SAVE: T     #S_SOFT; // Softwareschalter schreiben
NE3:  NOP   0;
NETWORK
TITLE =FC-Ausgang Q1

      U     #lb_Q1;
      =     #Q1;
NETWORK
TITLE =FC-Ausgang Q2

      U     #lb_Q2;
      =     #Q2;
NETWORK
TITLE =FC-ENO-Ausgang = Schaltausgang, für direkte FC-Verknüfpung

      O     #lb_Q1; // Ausgang 1
      O     #lb_Q2; // Ausgang 2
      SAVE  ; // auf FC-ENO-Ausgang geben
      CLR   ;

NETWORK
TITLE =Lokalen Speicher wieder in dauerhaften Zwischenspeicher

      L     LB     0;
      T     #bTmp;
      NOP   0;
END_FUNCTION

FUNCTION "m7b_udtCopyArray" : VOID
TITLE =kopiert einzelne UDT's von UDT-Arrays
//Kopiert UDT's aus Arrays, die Datenlänge des UDT wird automatisch ermittelt.
//Anpassungen der Datenlänge nach Änderungen an den UDT's entfällt somit.
//
//Achtung Array bzw. Speichergrenzen werden nicht überprüft.
//Gegebenenfalls, Indexangaben vorher auf Korrektheit prüfen bzw. limittieren!
//Bei inkorrekten Indexangaben geht CPU in STOP.
//
//Verwendung: Verwaltung von Datensätzen wie Rezepturen, Betriebsdaten,
//Positionsdaten usw. in der Steuerung.
//
//Kopiert wird von/zu: DB, statischen Lokaldaten im Instanz-DB
//(Multinnstanzfähig, ohne zus. Adresskorrektur, da Step7 bei Verwendung von
//Instanzdaten bei UDT's automatisch als Quelle [#84] DB und Nr. mit korrekter
//Adress angibt statt nur DI [#85])
//
//Nicht kopiert wrid von/zu lokalen Daten (TEMP), da vor- vorherige Lokaldaten
//benötigt werden (S7 aber nur vorherige Lokaldaten unterstützt)
//
//[IN]
//srcUdtArray : Anypointer auf den ersten UDT im Quell-Array
//srcIndex    : Index des Quell-UDT im Array, beginnend bei 0
//destUdtArray: Anypointer auf den ersten UDT im Ziel-Array
//destIndex   : Index des Ziel-UDT im Array, beginnend mit 0
//
//AUTOR: Stefan Maag, Dipl.-Ing. (FH) Elektrotechnik
//DATUM: 10/2007
//INTERNET: www.maagic7.de
//
//AENDERUNGSVERMERKE:
//--------------------------------------------------------------------------------
//DATUM        NAME       AENDERUNG
//--------------------------------------------------------------------------------
//20.03.2017   S.Maag     Verwendung von AR2 entfernt und Abfrage auf
//                        Daten Speicherbereich #87 vorheriger Lokaldatenstack
//                        hinzugefügt, da Daten aus vorherigem Stack nicht
//                        kopiert werden können, da BLKMOVE neuen L-Stack anlegt
//--------------------------------------------------------------------------------
//
AUTHOR : 'S.Maag'
FAMILY : Maagic7
VERSION : 0.1


VAR_INPUT
  srcUdtArray : ANY ;
  srcIndex : INT ;
  destUdtArray : ANY ;
  destIndex : INT ;
END_VAR
VAR_OUTPUT
  BLKMOV_RetVal : INT ;	//Return Value der Blockmovefunktion
END_VAR
VAR_TEMP
  pSRC : ANY ;	//mit Indexdaten modifizierter Quellpointer für BlockMove-Funktion
  pDEST : ANY ;	//mit Indexdaten modifizierter Zielpointer für BlockMove-Funktion
  dwPart1 : DWORD ;
  wPart2 : WORD ;
  dwPart3_Address : DWORD ;
  dwBitAddress : DWORD ;
  bMemory : BYTE ;	//Speicherbereich
END_VAR
BEGIN
NETWORK
TITLE =
//ANY
//Byte 0: 10h für S7
//Byte 1: Datentyp
//Byte 2..3: Wiederholungsfaktor
//Byte 4..5: DB-Nr
//Byte 6: Speicherbereich
//Byte 7..9: Byte/Bit-Adresse
//
//Speicherbereiche
//#80  P : Perepherie
//#81  E : Eingänge
//#82  A : Ausgänge
//#83  M : Merker
//#84  DB : Datenbaustein
//#85  DI : Instanz-DB
//#86  L  : Lokaldaten (L-Stack)
//#87  V  : Verherige Lokaldaten


NETWORK
TITLE =ANY-Pointer Quelle für BlockMove bearbeiten
//Beim Wiederholungsfaktor wird automatisch von Byte ausgegeangen.
//Für UDT's stimmt dies auch immer. Falls der Baustein allgemein zum kopieren von
//Anypointerbasierten Daten verwendet werden soll, so muss dies beachtet bzw.
//angepasst werden.
//Den ANY-Pointer Quelle mit den Indexdaten modifizieren und als ANY-Pointer für
//die BlockMove-Funktion speichern
      L     P##srcUdtArray; // Pointer auf den Quellpointer
      LAR1  ; // in Adressregister 1

      L     D [AR1,P#0.0]; // Part1
      T     #dwPart1;
      L     W [AR1,P#4.0]; // Part2
      T     #wPart2;
      L     D [AR1,P#6.0]; // Part3  (Address-Pointer)
      T     #dwPart3_Address;
      SRD   24; // Shift 3 Byte = Speicherbereich
      T     #bMemory;
      L     B#16#87; // Daten vom vorherigen Lockaldaten Stack (geht nicht!)
      ==I   ;
      SPB   ERR;


// Calculating the Address with Source ARRAY Index
      L     W [AR1,P#2.0]; // Wiederholungsfaktor
      L     #srcIndex;
      *I    ; // Offset aus Index für Quellbereich
      SLD   3; // ins Pointerformat konvertieren
      L     #dwPart3_Address; // Ursprüngliche Quelladdresse
      UD    DW#16#FFFFFF; // oberes Byte fuer Speicherbereich ausblenden
      +D    ; // Quelladresspointer mit verrechnetem Index
      T     #dwBitAddress;

      L     P##pSRC; // Pointer auf AnyPointer Quelle für BlockMove
      LAR1  ; // in Adressreguster 1

      L     #dwPart1; // Part 1 of ANY
      T     D [AR1,P#0.0]; // to pSRC [ANY]

      L     #wPart2; // Part 2
      T     W [AR1,P#4.0]; // DB-Nr.

      L     #dwPart3_Address; // Part 3 Address
      UD    DW#16#FF000000; // Speicherbereich maskieren
      L     #dwBitAddress; // mit Array-Index modifizierte Adresse
      OD    ; // Speicherbereich_Adresse zusammenführen
      T     D [AR1,P#6.0];

NETWORK
TITLE =ANY-Pointer Ziel für BlockMove bearbeiten

      L     P##destUdtArray; // Pointer auf den Quellpointer
      LAR1  ; // in Adressregister 1

      L     D [AR1,P#0.0]; // Part1
      T     #dwPart1;
      L     W [AR1,P#4.0]; // Part2
      T     #wPart2;
      L     D [AR1,P#6.0]; // Part3  (Address-Pointer)
      T     #dwPart3_Address;
      SRD   24; // Shift 3 Byte = Speicherbereich
      T     #bMemory;
      L     B#16#87; // Daten vom vorherigen Lockaldaten Stack (geht nicht!)
      ==I   ;
      SPB   ERR;

// Calculating the Address with Destination ARRAY Index
      L     W [AR1,P#2.0]; // Wiederholungsfaktor
      L     #destIndex;
      *I    ; // Offset aus Index für Quellbereich
      SLD   3; // ins Pointerformat konvertieren
      L     #dwPart3_Address; // Ursprüngliche Quelladdresse
      UD    DW#16#FFFFFF; // oberes Byte fuer Speicherbereich ausblenden
      +D    ; // Quelladresspointer mit verrechnetem Index
      T     #dwBitAddress;

      L     P##pDEST; // Pointer auf AnyPointer Quelle für BlockMove
      LAR1  ; // in Adressreguster 1

      L     #dwPart1; // Part 1 of ANY
      T     D [AR1,P#0.0]; // to pDEST [ANY]

      L     #wPart2; // Part 2
      T     W [AR1,P#4.0]; // DB-Nr.

      L     #dwPart3_Address; // Part 3 Address
      UD    DW#16#FF000000; // Speicherbereich maskieren
      L     #dwBitAddress; // mit Array-Index modifizierte Adresse
      OD    ; // Speicherbereich_Adresse zusammenführen
      T     D [AR1,P#6.0];

NETWORK
TITLE =kopieren der Daten mittels BlockMove

      CALL "BLKMOV" (
           SRCBLK                   := #pSRC,
           RET_VAL                  := #BLKMOV_RetVal,
           DSTBLK                   := #pDEST);
      NOP   0;
NETWORK
TITLE =

      SET   ;
      SAVE  ;
      BEA   ;

NETWORK
TITLE =
//Daten vom vorherigen Lokaldatenstack können nicht kopiert werden, da
//BLKMOVE neuen L-Stack öffnet und die Daten somit vom vor- vorherigen Stack
//wären
ERR:  L     W#16#8888; // Daten vom vorheriger Lockaldatenstack
      T     #BLKMOV_RetVal; // können nicht kopiert werden, da BLKMOVE neuen Stack anlegt
      SET   ;
      SAVE  ;
      BE    ;

END_FUNCTION

FUNCTION "m7b_MultiEventCounter" : VOID
TITLE =Multi-Ereigniszähler mit GesamtAnzahl im Ereignis 0
//Zähler für verschiedene Ereignisse. Es wird immer jeweils bei einem Zählvorgang
//der entsprechende Ereigniszähler und der Gesamtzähler erhöht. Eine Überprüfung
//auf die Gültigkeit des übergebenen DBs und richtige Länge wird nicht
//druchgeführt.
//
//AUTOR: Stefan Maag, Dipl.-Ing. (FH) Elektrotechnik
//DATUM: 5/2003
//INTERNET: www.maagic7.de
//
//AENDERUNGSVERMERKE:
//--------------------------------------------------------------------------------
//DATUM        NAME            AENDERUNG
//--------------------------------------------------------------------------------
//
//--------------------------------------------------------------------------------
//
//HINWEISE:
AUTHOR : 'S.Maag'
FAMILY : Maagic7
VERSION : 0.1


VAR_INPUT
  DBNr : INT ;	//Nr des Datenbausteins für Zählereignisse
  StartAdr : INT ;	//StartAdr. des ersten Eintrags
  EventNr : INT ;	//Nr des zu zählenden Ereignisses; Nr.0 = Gesamtzaehler
  Count : BOOL ;	//Befehl zählen
END_VAR
VAR_TEMP
  tmpDB : INT ;
  tmpPtrOff : INT ;
  AR1 : DWORD ;
END_VAR
BEGIN
NETWORK
TITLE =Überprüfung auf Zählen!

      UN    #Count;
      BEB   ;
NETWORK
TITLE =ungültige EreignisNr - ENDE

      L     #EventNr;
      L     1;
      <I    ;
      BEB   ;
NETWORK
TITLE =DB öffnen und Pointer auf StartAdresse erzeugen

      TAR1  #AR1; // Adressregister 1 sichern

      L     #DBNr;
      T     #tmpDB;

      AUF   DB [#tmpDB];

      L     #StartAdr; // Startadresse ins Pointerformat
      SLD   3;
      TAR1  ; // ins Adressregister 1

NETWORK
TITLE =GesamtZaehler bearbeiten


      L     DBD [AR1,P#0.0]; // Gesamtzählerstand aus DB lesen
      +     1;
      T     DBD [AR1,P#0.0]; // neuen Gesamtzählerstand speichern

NETWORK
TITLE =Pointer Auf EreignisZähler-Daten erzeugen

      TAR1  ; // Pointer auf Startadresse in Akku 1 zurueck
      L     #EventNr; // EreignisNr
      SLD   5; // EreignisNr -> BitPointer (*16; DINT=32Bit)
      +D    ; // Pointer aus Ereignis zum StartPointer addieren
      LAR1  ; // Pointer auf EreignisZähler nach Adressregister 1

NETWORK
TITLE =EreignisZähler bearbeiten

      L     DBD [AR1,P#0.0]; // Ereigniszählerstand aus DB lesen
      +     1;
      T     DBD [AR1,P#0.0]; // neuen Ereigniszählerstand speichern

NETWORK
TITLE =FC-ENO Ausgang

      LAR1  #AR1; // ursprüngliches Adressregister 1 herstellen
      SET   ;
      SAVE  ;
      CLR   ;

END_FUNCTION

FUNCTION "m7b_udtCompareArray" : VOID
TITLE =udt Daten in Arrays vergleichen
//Vergleicht UDT's aus Arrays, die Datenlänge des UDT wird automatisch ermittelt.
//Anpassungen der Datenlänge nach Änderungen an den UDT's entfällt somit.
//
//Achtung!
//   Array bzw. Speichergrenzen werden nicht überprüft.
//   Gegebenenfalls, Indexangaben vorher auf Korrektheit prüfen bzw. limittieren!
//   Bei inkorrekten Indexangaben geht CPU in STOP.
//
//   Bei Verwendung von Strings in UDT's kann es vorkommen, dass zwischen dem
//   letzten Zeichen und reservierter Stringlänge noch tote Bytes mit
//   undefinierten Werten liegen. Dann ergibt der Vergleich des UDT ungleich, ein
//   Stringvergleich würde jedoch gleich ergeben.
//
//Verwendung: Verwaltung von Datensätzen wie Rezepturen, Betriebsdaten,
//Positionsdaten usw. in der Steuerung.
//
//[IN]
//srcUdtArray : Anypointer auf den ersten UDT im Quell-Array
//srcIndex    : Index des Quell-UDT im Array, beginnend bei 0
//cmpUdtArray : Anypointer auf den ersten UDT im Vergleichs-Array
//cmpIndex    : Index des Vergleichs-UDT im Array, beginnend mit 0
//
//[RET]
//ENO         : True if datas are equal
//
//AUTOR: Stefan Maag, Dipl.-Ing. (FH) Elektrotechnik
//DATUM: 10/2010
//INTERNET: www.maagic7.de
//
//AENDERUNGSVERMERKE:
//--------------------------------------------------------------------------------
//DATUM        NAME            AENDERUNG
//--------------------------------------------------------------------------------
//
//--------------------------------------------------------------------------------
//
//HINWEISE: AR2, Global- und Instanz DB muessen nicht gesichert werden, da diese
//           bei Call Aufrufen automatisch vom System wieder hergestellt werden.
//          (Bei UC Aufrufen nicht!)
//
//Vergleichroutine basiert auf m7b_DB_COMPARE_ByRef FC218
AUTHOR : 'S.Maag'
FAMILY : Maagic7
VERSION : 0.1


VAR_INPUT
  srcUdtArray : ANY ;
  srcIndex : INT ;
  cmpUdtArray : ANY ;
  cmpIndex : INT ;
END_VAR
VAR_TEMP
  AR1 : DWORD ;
  p_srcData : DWORD ;
  p_cmpData : DWORD ;
  srcRepeat : WORD ;
  cmpRepeat : WORD ;
  srcDataType : BYTE ;
  cmpDataType : BYTE ;
  srcDB_No : WORD ;
  cmpDB_no : WORD ;
  DB_NO : WORD ;
  srcSpeicherBereich : BYTE ;
  cmpSpeicherBereich : BYTE ;
  LOOPS : INT ;
  NoOfBytes : INT ;
  srcIsDB : BOOL ;
  cmpIsDB : BOOL ;
  pTest : DWORD ;
END_VAR
BEGIN
NETWORK
TITLE =Adressregiste 1 sichern
//Adressregister 2 Global- und Instanz DB werden bei CALL-Aufrufen automatisch
//vom System gesichert, bei UC nicht!
      TAR1  #AR1; // Adressregister 1 sichern

NETWORK
TITLE =Adressdaten aus ANY-Pointer extrahieren
//Beim Wiederholungsfaktor wird automatisch von Byte ausgegeangen.
//Für UDT's stimmt dies auch immer. Falls der Baustein allgemein zum vergleichen
//von Anypointerbasierten Daten verwendet werden soll, so muss dies beachtet bzw.
//angepasst werden.
//
      L     P##srcUdtArray; // Pointer auf den Quellpointer
      LAR1  ; // in Adressregister 1

      L     B [AR1,P#1.0]; // Byte 1 = Datentyp
      T     #srcDataType;

      L     B [AR1,P#6.0]; // Byte 6 = Speicherbereich
      T     #srcSpeicherBereich;

      L     W [AR1,P#4.0]; // DB-Nummer oder 0, wenn kein DB
      T     #srcDB_No;

      L     W [AR1,P#2.0]; // Wiederholungsfaktor
      T     #srcRepeat;
      L     #srcIndex;
      *I    ; // Offset aus Index für Quellbereich
      SLD   3; // ins Pointerformat konvertieren
      L     D [AR1,P#6.0]; // DatenAdresse im Pointeformat aus ANY
      +D    ; // Adresspointer mit verrechnetem Index
      T     #p_srcData; // Pointer Source Data

      L     P##cmpUdtArray; // Pointer auf Vergleichs UDT
      LAR1  ; // in Adressregister 1

      L     B [AR1,P#1.0]; // Byte 1 = Datentyp
      T     #cmpDataType;

      L     B [AR1,P#6.0]; // Byte 6 = Speicherbereich
      T     #cmpSpeicherBereich;

      L     W [AR1,P#4.0]; // DB-Nummer oder 0, wenn kein DB
      T     #cmpDB_no;

      L     W [AR1,P#2.0]; // Wiederholungsfaktor
      T     #cmpRepeat;
      L     #cmpIndex;
      *I    ; // Offset aus Index für Vergleichsbereich
      SLD   3; // ins Pointerformat konvertieren
      L     D [AR1,P#6.0]; // DatenAdresse im Pointeformat aus ANY
      +D    ; // Adresspointer mit verrechnetem Index
      T     #p_cmpData; // Pointer Vergleichsdaten

NETWORK
TITLE =Prüfen ob gleiches Datenformat, wenn NEIN, dann Daten ungleich
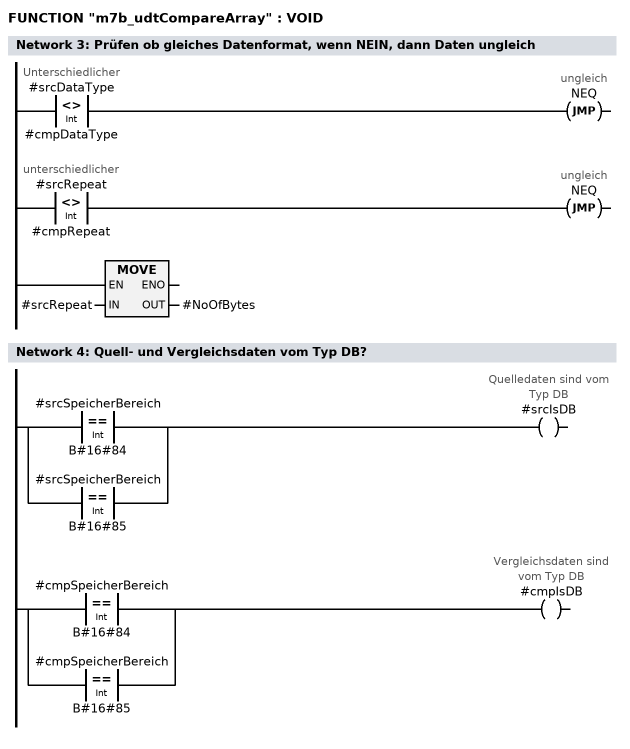

      L     #srcDataType; // Unterschiedlicher
      L     #cmpDataType; // Datentyp?
      <>I   ;
      SPB   NEQ; // ungleich

      L     #srcRepeat; // unterschiedlicher
      L     #cmpRepeat; // Wiederholungsfaktor
      <>I   ;
      SPB   NEQ; // ungleich

      L     #srcRepeat; // srcRepeat=cmpRepeat, deshalb
      T     #NoOfBytes; // Anzahl zu vergleichender Bytes gleich

NETWORK
TITLE =Quell- und Vergleichsdaten vom Typ DB?

      O(    ;
      L     #srcSpeicherBereich;
      L     B#16#84; // Datenbaustein
      ==I   ;
      )     ;
      O(    ;
      L     #srcSpeicherBereich;
      L     B#16#85; // Instanzdatenbaustein
      ==I   ;
      )     ;
      =     #srcIsDB; // Quelledaten sind vom Typ DB

      O(    ;
      L     #cmpSpeicherBereich;
      L     B#16#84; // Datenbaustein
      ==I   ;
      )     ;
      O(    ;
      L     #cmpSpeicherBereich;
      L     B#16#85; // Instanzdatenbaustein
      ==I   ;
      )     ;
      =     #cmpIsDB; // Vergleichsdaten sind vom Typ DB

NETWORK
TITLE =Vorbereitung für Vergleichsroutine
//Für die eigentliche Vergleichsroutine ist es nur relevant ob die Daten aus
//einem DB stammen, nicht ob Instanz oder Global-DB. Für den vergleich wird
//temporär immer ein DB als Global-DB, der andere als Instanz-DB geöffnet. Da dies
// nur nach Nummern geschieht, ist es egal welcher der DBs wie geöffnet wird.
//Codierung Speicherbereich:
//80h : P : Peripherie
//81h : E : Eingänge
//82h : A : Ausgänge
//83h : M : Merker
//84h : DB: Datenbaustein
//85h : DI: Instanzdatenbaustein
//86h : L : Lokaldaten (L-Stack)
//87h : V : voriger Lokaldatenstack
      UN    #srcIsDB; // Wenn weder Qell noch Vergleichsdaten
      UN    #cmpIsDB; // vom Typ DB
      SPB   DO; // dann keine Modifikation der DB-Kennung nötig, sofort vergleichen

      UN    #srcIsDB; // Wenn Quell-Daten nicht aus DB dann weiter,
      SPB   w1; // sonst Global-DB Kennung in Quelldatenpointer eintragen

      LAR1  P##p_srcData; // Adressregister 1 mit Pointer auf p_srcData laden
      L     B#16#84; // Wert für Global-DB-Kennung
      T     B [AR1,P#0.0]; // 84h=DB in p_srcData als Speicherbereichskennung eintragen

      AUF   DB [#srcDB_No]; // Datenbaustein Quelldaten als Global-DB öffnen

w1:   UN    #cmpIsDB; // Wenn Vergleichs-Daten nicht aus DB dann weiter,
      SPB   save; // sonst Instanz-DB Kennung in Quelldatenpointer eintragen

      LAR1  P##p_cmpData; // Adressregister 1 mit Pointer auf p_cmpData laden
      L     B#16#85; // Wert für Instanz-DB-Kennung
      T     B [AR1,P#0.0]; // 85h=DB in p_srcData als Speicherbereichskennung eintragen

      AUF   DI [#cmpDB_no]; // Datenbaustein Vergleichsdaten als Instanz-DB öffnen

save: L     #p_srcData; // Pointer der Quelldaten p_srcData in Adressregister 1
      LAR1  ;
      L     #p_cmpData; // Pointer der Vergleichsdaten p_cmpData in Adressregister 2
      LAR2  ;
NETWORK
TITLE =Vergleich der Daten
//Vergleich der Daten
//Vergleichroutine basiert auf m7b_DB_COMPARE_ByRef FC218
DO:   L     #NoOfBytes; // Anzahl der zu vergleichenden Bytes
      L     4; // in Anzahl der 32-Bit-Werte umrechen
      /I    ;
      SPZ   bts; // Wenn 0 32-Bit Werte, dann weiter mit letzten 3 Bytes
LOOP: T     #LOOPS;
      L     D [AR1,P#0.0]; // QuellDaten lesen
      L     D [AR2,P#0.0]; // VergleichsDaten lesen
      <>D   ; // wenn nicht gleich, dann Ende
      SPB   NEQ;
      +AR1  P#4.0; // Quell-Pointer in AR1 um 4 Bytes erhöhen
      +AR2  P#4.0; // Vergleichs-Pointer in AR2 um 4 Bytes erhöhen
      L     #LOOPS; // Schleifenzähler wieder in Akku 1 zurück
      LOOP  LOOP; // Schleifenzähler bearbeiten

bts:  L     #NoOfBytes; // nun noch die evtl. letzte 3 Bytes prüfen
      L     2#11; // Anzahl übriger Bytes maskieren
      UW    ; // Anzahl übriger Bytes
      SPZ   EQ; // Wenn 0 dann ENDE
LOP1: T     #LOOPS;
      L     B [AR1,P#0.0]; // QuellDaten lesen
      L     B [AR2,P#0.0]; // VergleichsDaten lesen
      <>I   ; // wenn nicht gleich, dann Ende
      SPB   NEQ;
      +AR1  P#1.0; // Quell-Pointer in AR1 um 1 Bytes erhöhen
      +AR2  P#1.0; // Vergleichs-Pointer in AR2 um 1 Bytes erhöhen
      L     #LOOPS; // Schleifenzähler wieder in Akku 1 zurück
      LOOP  LOP1; // Schleifenzähler bearbeiten

EQ:   SET   ; // Daten sind gleich (equal)
      SAVE  ;
      CLR   ;
      SPA   END;

NEQ:  CLR   ; // Daten sind ungleich (not equal)
      SAVE  ;

NETWORK
TITLE =Adressregister 1 wieder herstellen

END:  LAR1  #AR1; // ursprüngliches Adressregister 1 herstellen


END_FUNCTION

FUNCTION "m7b_2xSTART_SWITCH" : VOID
TITLE =2-fach Startumschalter
//Dieser Baustein ermöglicht, 2 Geräte (z.B. Kompressoren) abwechselnd
//einzuschalten. Dazu werden bei jedem Ausschalten eines Gerätes die beiden
//FRG-Ausgänge des Bausteins umgeschaltet.
//
//Verwendung: Startumschaltung von Kompressorenpaaren bei Klimaanlagen
//
//AUTOR: Stefan Maag, Dipl.-Ing. (FH) Elektrotechnik
//DATUM: 4/2004
//INTERNET: www.maagic7.de
//
//AENDERUNGSVERMERKE:
//--------------------------------------------------------------------------------
//DATUM        NAME            AENDERUNG
//--------------------------------------------------------------------------------
//
//--------------------------------------------------------------------------------
//
//HINWEISE:
AUTHOR : 'S.Maag'
FAMILY : Maagic7
VERSION : 0.1


VAR_INPUT
  G1_RUN : BOOL ;	//Eingang Gerät 1 läuft
  G2_RUN : BOOL ;	//Eingang Gerät 2 läuft
END_VAR
VAR_OUTPUT
  FRG1 : BOOL ;	//Freigabe Start Gerät 1
  FRG2 : BOOL ;	//Freigabe Start Gerät 2
END_VAR
VAR_IN_OUT
  bTMP : BYTE ;	//statisches Hilfsbyte
END_VAR
VAR_TEMP
  lb_SWITCH : BOOL ;	//Bit 0 von IO-Byte bTMP : Umschalter
  lb_FN : BOOL ;	//Negative Flanke Geräte ausgeschaltet
  lb2 : BOOL ;
  lb3 : BOOL ;
  lb4 : BOOL ;
  lb5 : BOOL ;
  lb6 : BOOL ;
  lb7 : BOOL ;	//Bit 7 von IO-Byte bTMP
END_VAR
BEGIN
NETWORK
TITLE =statisches HilfsByte in Lokaldatenbereich

      L     #bTMP;
      T     LB     0;
      NOP   0;
NETWORK
TITLE =Freigabe umschalten, wenn beide Geräte aus sind

      O     #G1_RUN;
      O     #G2_RUN;
      FN    #lb_FN;
      SPBN  NE2;
      UN    #lb_SWITCH;
      =     #lb_SWITCH;
NE2:  NOP   0;
NETWORK
TITLE =Bausteinausgang Freigabe Gerät 1

      UN    #lb_SWITCH;
      =     #FRG1;

NETWORK
TITLE =Bausteinausgang Freigabe Gerät 2

      U     #lb_SWITCH;
      =     #FRG2;

NETWORK
TITLE =statisches HilfsByte aus Lokaldatenbereich zurück

      L     LB     0;
      T     #bTMP;
      NOP   0;
NETWORK
TITLE =

      SET   ;
      SAVE  ;
      CLR   ;


END_FUNCTION

FUNCTION "m7b_MSG_2_ML" : VOID
TITLE =Meldungen (16Stk) mittels 2er Meldeleuchten anzeigen
//AUTOR: Stefan Maag, Dipl.-Ing. (FH) Elektrotechnik
//DATUM: 04/2006
//INTERNET: www.maagic7.de
//
//AENDERUNGSVERMERKE:
//--------------------------------------------------------------------------------
//DATUM        NAME      AENDERUNG
//--------------------------------------------------------------------------------
//
//--------------------------------------------------------------------------------
//
//HINWEISE:
AUTHOR : 'S.Maag'
FAMILY : Maagic7
VERSION : 0.1


VAR_INPUT
  MSG_1_8 : BYTE ;	//Meldung 1 bis 8 als Bits
  MSG_9_16 : BYTE ;
  TAKT_BYTE : BYTE ;	//System Taktmerkerbyte
END_VAR
VAR_OUTPUT
  ML1 : BOOL ;
  ML2 : BOOL ;
END_VAR
VAR_TEMP
  MSG_1 : BOOL ;
  MSG_2 : BOOL ;
  MSG_3 : BOOL ;
  MSG_4 : BOOL ;
  MSG_5 : BOOL ;
  MSG_6 : BOOL ;
  MSG_7 : BOOL ;
  MSG_8 : BOOL ;
  MSG_9 : BOOL ;
  MSG_10 : BOOL ;
  MSG_11 : BOOL ;
  MSG_12 : BOOL ;
  MSG_13 : BOOL ;
  MSG_14 : BOOL ;
  MSG_15 : BOOL ;
  MSG_16 : BOOL ;
  TAKT_100 : BOOL ;
  TAKT_200 : BOOL ;
  TAKT_400 : BOOL ;
  TAKT_500 : BOOL ;
  TAKT_800 : BOOL ;
  TAKT_1000 : BOOL ;
  TAKT_1600 : BOOL ;
  TAKT_2000 : BOOL ;
END_VAR
BEGIN
NETWORK
TITLE =Meldungsbits für Einzelbitverarbeitung in Lokaldatenbereich

      L     #MSG_1_8;
      T     LB     0;

      L     #MSG_9_16;
      T     LB     1;

      L     #TAKT_BYTE;
      T     LB     2;

      L     LW     0; // Alle 16 Meldungsbits laden
      L     0; // und auf 0 prüfen
      ==I   ; // wenn 0, dann keine Meldung
      SPB   E0; // keine Meldung

NETWORK
TITLE =Meldung nach Priorität auswählen
//Durch vertauschen der Auswertungen und Sprünge kann die Priortät der
//angezeigten Meldungen in gewünschter Reihenfolge festgelegt werden
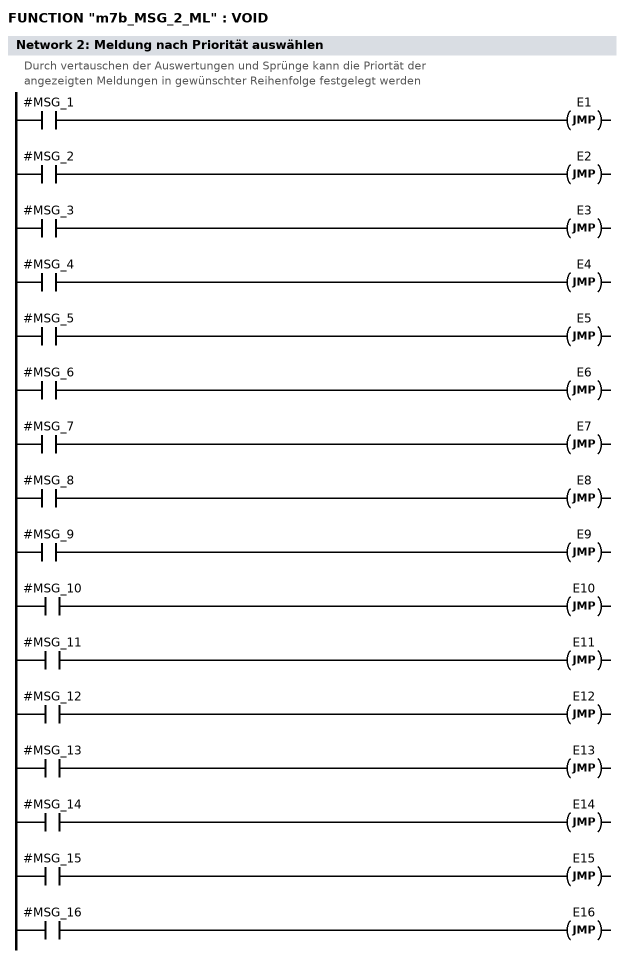
      U     #MSG_1;
      SPB   E1;
      U     #MSG_2;
      SPB   E2;
      U     #MSG_3;
      SPB   E3;
      U     #MSG_4;
      SPB   E4;
      U     #MSG_5;
      SPB   E5;
      U     #MSG_6;
      SPB   E6;
      U     #MSG_7;
      SPB   E7;
      U     #MSG_8;
      SPB   E8;
      U     #MSG_9;
      SPB   E9;
      U     #MSG_10;
      SPB   E10;
      U     #MSG_11;
      SPB   E11;
      U     #MSG_12;
      SPB   E12;
      U     #MSG_13;
      SPB   E13;
      U     #MSG_14;
      SPB   E14;
      U     #MSG_15;
      SPB   E15;
      U     #MSG_16;
      SPB   E16;

NETWORK
TITLE =Meldungen 0..3: ML2=AUS

E0:   CLR   ; // keine Störung
      =     #ML1;
      SPA   M0;

E1:   U     #TAKT_1000;
      =     #ML1;
      SPA   M0;

E2:   U     #TAKT_400;
      =     #ML1;
      SPA   M0;

E3:   SET   ;
      =     #ML1;

M0:   CLR   ;
      =     #ML2;
      SPA   END;

NETWORK
TITLE =Meldungen 4..7: ML2=TAKT_400ms

E4:   CLR   ;
      =     #ML1;
      SPA   M1;

E5:   U     #TAKT_1000;
      =     #ML1;
      SPA   M1;

E6:   U     #TAKT_400;
      =     #ML1;
      SPA   M1;

E7:   SET   ;
      =     #ML1;

M1:   U     #TAKT_1000;
      =     #ML2;
      SPA   END;

NETWORK
TITLE =Meldungen 8..11: ML2=TAKT_1000ms

E8:   CLR   ;
      =     #ML1;
      SPA   M2;

E9:   U     #TAKT_1000;
      =     #ML1;
      SPA   M2;

E10:  U     #TAKT_400;
      =     #ML1;
      SPA   M2;

E11:  SET   ;
      =     #ML1;

M2:   U     #TAKT_400;
      =     #ML2;
      SPA   END;

NETWORK
TITLE =Meldungen 12..15: ML2=EIN

E12:  CLR   ;
      =     #ML1;
      SPA   M3;

E13:  U     #TAKT_1000;
      =     #ML1;
      SPA   M3;

E14:  U     #TAKT_400;
      =     #ML1;
      SPA   M3;

E15:  SET   ;
      =     #ML1;

M3:   SET   ;
      =     #ML2;
NETWORK
TITLE =Meldung 16: Beide Lampen blinken abwechselnd

E16:  U     #TAKT_1000;
      =     #ML1;
      UN    #TAKT_1000;
      =     #ML2;

NETWORK
TITLE =

END:  BEA   ;

END_FUNCTION

FUNCTION "m7b_4SensorSpeed" : VOID
TITLE =Geschwindigkeit Achse mit 4 Sensoren bremsen/Endstellung - vw/rw
//Geschwindigkeit Achse mit 4 Sensoren
//  - Endstellung vorwärts
//  - Bremsen vorwärts
//  - Bremsen rückwärts
//  - Endstellung rückwärts
//
//Das Signal der Bremssensoren wird gemerkt, sie können also überfahren werden.
//Dies ist unbedingt notwendig bei Verwendung von Zylindersensoren.
//
//ACHTUNG: Um ein ungewollt schnelles losfahren zu vermeiden, ist es
//empfehlenswert, bei Not-Aus, den RESET auszulösen.
//Somit wird beim ersten Start dann langsam gefahren, bis ein Sensor explizit
//wieder schnelle Geschwindigkeit erlaubt.
//
//[IN]
//vw        : Richtung vorwärts ist aktiv
//rw        : Richtung rückwärts ist aktiv
//EST_vw    : Sensor Endstellung vorwärts
//BREMS_vw  : Sensor Bremsen vorwärts
//BREMS_rw  : Sensor Bremsen rückwärts
//EST_rw    : Sensor Endstellung rückwärts
//RESET     : Schnellmerker löschen (z.B. bei Not-Aus & CPU-RESTART)
//
//[OUT]
//vw_schnell : Achse vorwärts schnelle Geschwindigkeit
//rw_schnell : Achse rückwärts schnelle Geschwindigkeit
//
//[IN_OUT]
//bTmp : exterenes Hilfbyte zur Datenspeicherung
//
//AUTOR: Stefan Maag, Dipl.-Ing. (FH) Elektrotechnik
//DATUM: 2/2006
//INTERNET: www.maagic7.de
//
//AENDERUNGSVERMERKE:
//--------------------------------------------------------------------------------
//DATUM        NAME        AENDERUNG
//--------------------------------------------------------------------------------
//03.12.2008   S.Maag     Änderung der Ausgänge von langsam nach schnell, und
//                        zusätzlicher RESET-Eingang zum löschen der Schnell-
//                        Befehle, das hat den Vorteil, dass man verhindern kann,
//                        dass bei einem Neustart ohne belegte Sensoren ungewollt
//                        schnell losgefahren wird.
//--------------------------------------------------------------------------------
//
//HINWEISE:
AUTHOR : 'S.Maag'
FAMILY : Maagic7
VERSION : 0.1


VAR_INPUT
  vw : BOOL ;	//Richtung vorwärts aktiv
  rw : BOOL ;	//Richtung rückwärts aktiv
  EST_vw : BOOL ;	//Sensor Enstellung vorwärts
  BREMS_vw : BOOL ;	//Sensor Bremsen Endstellung vorwärts
  BREMS_rw : BOOL ;	//Sensor Bremsen Enstellung rückwärts
  EST_rw : BOOL ;	//Sensor Endstellung rückwärts
  RESET : BOOL ;	//Rücksetzten der Schnellbefehle, z.B. bei CPU-Restart
END_VAR
VAR_OUTPUT
  vw_schnell : BOOL ;
  rw_schnell : BOOL ;
END_VAR
VAR_IN_OUT
  bTmp : BYTE ;	//Hilfbyte für Signalspeicherung
END_VAR
VAR_TEMP
  lb_schnell_vw : BOOL ;	//Lokaler Speicher: schnell vorwärts
  lb_schnell_rw : BOOL ;	//Lokaler Speicher: schnell rückwärts
  lb_FN_BREMS_vw : BOOL ;	//Lokaler Speicher: negative Flanke Sensor Bremsen vorwärts
  lb_FN_BREMS_rw : BOOL ;	//Lokaler Speicher: negative Flanke Sensor Bremsen rückwärts
  lb4 : BOOL ;	//Lokaler Speicher
  lb5 : BOOL ;	//Lokaler Speicher
  lb6 : BOOL ;	//Lokaler Speicher
  lb7 : BOOL ;	//Lokaler Speicher
END_VAR
BEGIN
NETWORK
TITLE =Dauerhaften Zwischenspeicher in Lokaldatenbereich
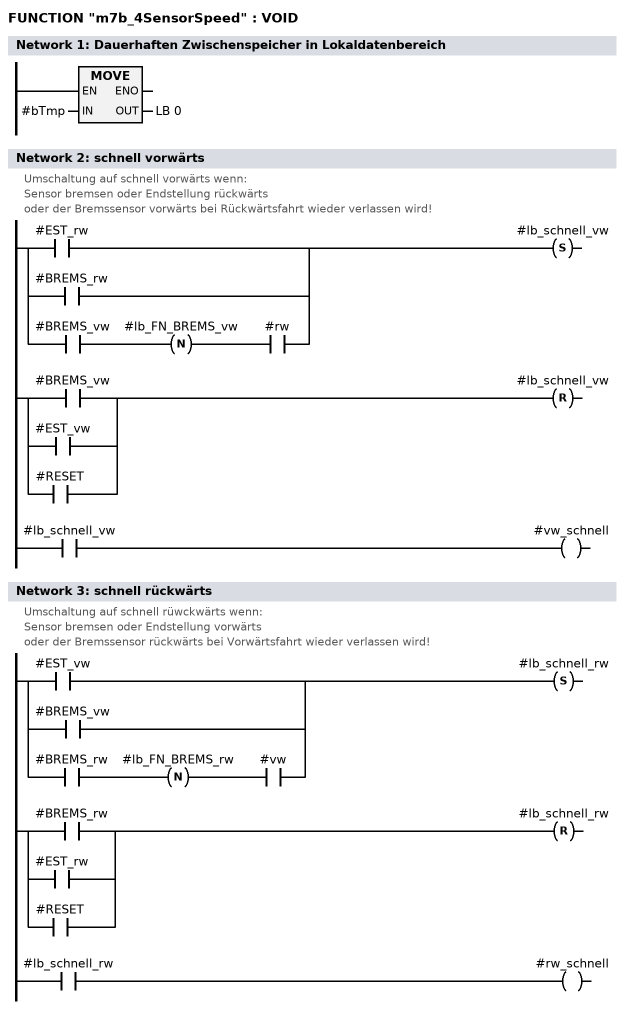

      L     #bTmp;
      T     LB     0;
      NOP   0;
NETWORK
TITLE =schnell vorwärts
//Umschaltung auf schnell vorwärts wenn:
//Sensor bremsen oder Endstellung rückwärts
//oder der Bremssensor vorwärts bei Rückwärtsfahrt wieder verlassen wird!
      U(    ;
      O     #EST_rw;
      O     #BREMS_rw;
      O(    ;
      U     #BREMS_vw;
      FN    #lb_FN_BREMS_vw;
      U     #rw;
      )     ;
      )     ;
      S     #lb_schnell_vw;
      U(    ;
      O     #BREMS_vw;
      O     #EST_vw;
      O     #RESET;
      )     ;
      R     #lb_schnell_vw;
      U     #lb_schnell_vw;
      =     #vw_schnell;
NETWORK
TITLE =schnell rückwärts
//Umschaltung auf schnell rüwckwärts wenn:
//Sensor bremsen oder Endstellung vorwärts
//oder der Bremssensor rückwärts bei Vorwärtsfahrt wieder verlassen wird!
      U(    ;
      O     #EST_vw;
      O     #BREMS_vw;
      O(    ;
      U     #BREMS_rw;
      FN    #lb_FN_BREMS_rw;
      U     #vw;
      )     ;
      )     ;
      S     #lb_schnell_rw;
      U(    ;
      O     #BREMS_rw;
      O     #EST_rw;
      O     #RESET;
      )     ;
      R     #lb_schnell_rw;
      U     #lb_schnell_rw;
      =     #rw_schnell;
NETWORK
TITLE =FC-ENO-Ausgang

      O     #lb_schnell_vw;
      O     #lb_schnell_rw;
      SAVE  ;
      CLR   ;

NETWORK
TITLE =Lokalen Speicher wieder in dauerhaften Zwischenspeicher

      L     LB     0;
      T     #bTmp;
      NOP   0;
END_FUNCTION

FUNCTION "m7b_2SensorSpeed" : VOID
TITLE =Geschwindigkeit Achse mit 2 mitfahrenden Sensoren
//Geschwindigkeit Achse mit 2 mitfahrenden Sensoren
//  - Sensor vorw.  (voraus bei vorwärts)
//  - Sensor rückw. (voraus bei rückwärts)
//
//Das Signal der Sensoren wird gemerkt, sie können also überfahren werden.
//
//[IN]
//vw        : Richtung vorwärts ist aktiv
//rw        : Richtung rückwärts ist aktiv
//SENS_vw   : Sensor in Vorwärtsrichtung
//SENS_rw   : Sensor in Rückwärtsrichtung
//
//[OUT]
//STOP_vw    : Stop, Endstellung vorwärts
//Bremsen_vw : Achse vorwärts langsame Geschwindigkeit (bremsen)
//Bremsen_rw : Achse rückwärts langsame Geschwindigkeit (bremsen)
//STOP_rw    : Stop, Endstellung rückwärts
//
//[IN_OUT]
//bTmp : exterenes Hilfbyte zur Datenspeicherung
//
//AUTOR: Stefan Maag, Dipl.-Ing. (FH) Elektrotechnik
//DATUM: 2/2006
//INTERNET: www.maagic7.de
//
//AENDERUNGSVERMERKE:
//--------------------------------------------------------------------------------
//DATUM        NAME            AENDERUNG
//--------------------------------------------------------------------------------
//
//--------------------------------------------------------------------------------
//
//HINWEISE:
AUTHOR : 'S.Maag'
FAMILY : Maagic7
VERSION : 0.1


VAR_INPUT
  vw : BOOL ;	//Richtung vorwärts aktiv
  rw : BOOL ;	//Richtung rückwärts aktiv
  SENS_vw : BOOL ;	//Sensor Bremsen Endstellung vorwärts
  SENS_rw : BOOL ;	//Sensor Bremsen Enstellung rückwärts
END_VAR
VAR_OUTPUT
  STOP_vw : BOOL ;	//Stop vorwärts
  Bremsen_vw : BOOL ;	//Bremsen vorwaerts
  Bremsen_rw : BOOL ;	//Bremsen rückwärts
  STOP_rw : BOOL ;	//Stop rückwärts
END_VAR
VAR_IN_OUT
  bTmp : BYTE ;	//Hilfbyte für Signalspeicherung
END_VAR
VAR_TEMP
  lb_STOP_vw : BOOL ;	//Lokaler Speicher: Stop vorwärts, Endstellung
  lb_bremsen_vw : BOOL ;	//Lokaler Speicher: Bremsen vorwärts
  lb_bremsen_rw : BOOL ;	//Lokaler Speicher: Bremsen rückwärts
  lb_STOP_rw : BOOL ;	//Lokaler Speicher: Stop rückwärts, Endstellung
  lb_FP_SENS_vw : BOOL ;	//Lokaler Speicher: positive Flanke Sensor vorwärts
  lb_FP_SENS_rw : BOOL ;	//Lokaler Speicher: positive Flanke Sensor rückwärts
  lb_FN_SENS_vw : BOOL ;	//Lokaler Speicher: negative Flanke Sensor vorwärts
  lb_FN_SENS_rw : BOOL ;	//Lokaler Speicher: negative Flanke Sensor rückwärts
  FP_SENS_vw : BOOL ;
  FP_SENS_rw : BOOL ;
  FN_SENS_vw : BOOL ;
  FN_SENS_rw : BOOL ;
END_VAR
BEGIN
NETWORK
TITLE =Dauerhaften Zwischenspeicher in Lokaldatenbereich
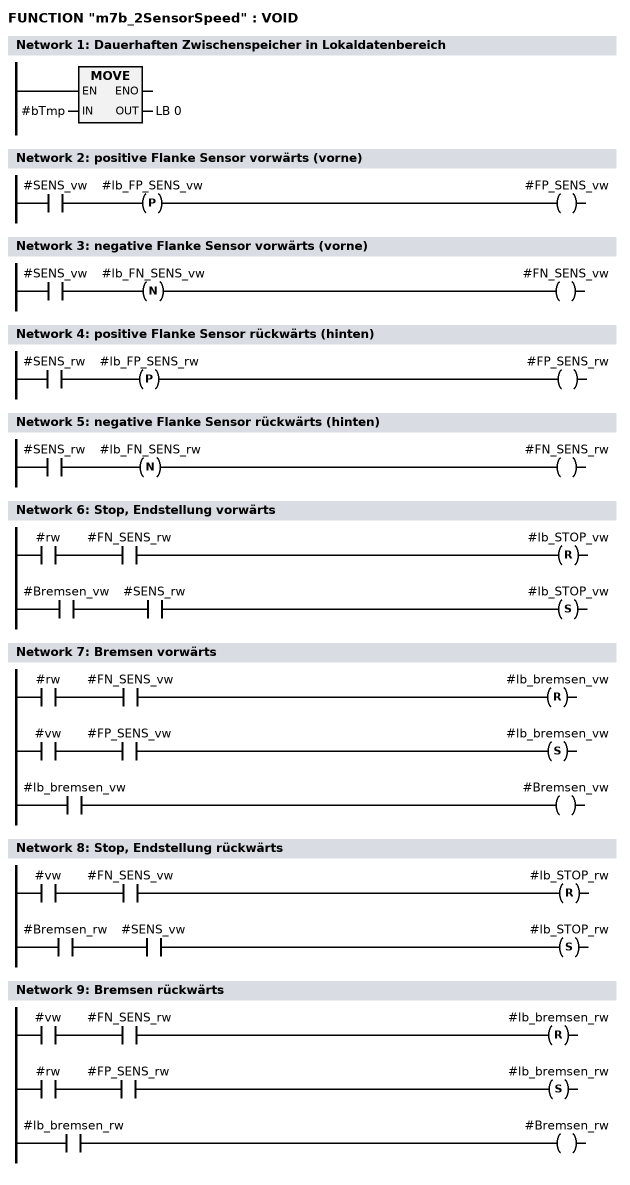

      L     #bTmp;
      T     LB     0;
      NOP   0;
NETWORK
TITLE =positive Flanke Sensor vorwärts (vorne)

      U     #SENS_vw;
      FP    #lb_FP_SENS_vw;
      =     #FP_SENS_vw;
NETWORK
TITLE =negative Flanke Sensor vorwärts (vorne)

      U     #SENS_vw;
      FN    #lb_FN_SENS_vw;
      =     #FN_SENS_vw;
NETWORK
TITLE =positive Flanke Sensor rückwärts (hinten)

      U     #SENS_rw;
      FP    #lb_FP_SENS_rw;
      =     #FP_SENS_rw;
NETWORK
TITLE =negative Flanke Sensor rückwärts (hinten)

      U     #SENS_rw;
      FN    #lb_FN_SENS_rw;
      =     #FN_SENS_rw;
NETWORK
TITLE =Stop, Endstellung vorwärts

      U     #rw;
      U     #FN_SENS_rw;
      R     #lb_STOP_vw;
      U     #Bremsen_vw;
      U     #SENS_rw;
      S     #lb_STOP_vw;
      NOP   0;
NETWORK
TITLE =Bremsen vorwärts

      U     #rw;
      U     #FN_SENS_vw;
      R     #lb_bremsen_vw;
      U     #vw;
      U     #FP_SENS_vw;
      S     #lb_bremsen_vw;
      U     #lb_bremsen_vw;
      =     #Bremsen_vw;
NETWORK
TITLE =Stop, Endstellung rückwärts

      U     #vw;
      U     #FN_SENS_vw;
      R     #lb_STOP_rw;
      U     #Bremsen_rw;
      U     #SENS_vw;
      S     #lb_STOP_rw;
      NOP   0;
NETWORK
TITLE =Bremsen rückwärts

      U     #vw;
      U     #FN_SENS_rw;
      R     #lb_bremsen_rw;
      U     #rw;
      U     #FP_SENS_rw;
      S     #lb_bremsen_rw;
      U     #lb_bremsen_rw;
      =     #Bremsen_rw;
NETWORK
TITLE =FC-ENO-Ausgang

      O     #lb_bremsen_vw;
      O     #lb_bremsen_rw;
      SAVE  ;
      CLR   ;

NETWORK
TITLE =Lokalen Speicher wieder in dauerhaften Zwischenspeicher

      L     LB     0;
      T     #bTmp;
      NOP   0;
END_FUNCTION

FUNCTION "m7b_SoftEncoder" : VOID
TITLE =SoftEncoder mit Sensor
//SoftEncoder mit Sensor
//Software-Encoder mit Sensor und Richtungssignal erzeugen
//
//VERWENDUNG:
//Für Standard 4 Puls Schrauben-Encoder von Transporttischen
//
//[IN]
//SENSOR    Encodersignal, Sensor
//POS       Richtungssignal positiv / Transport vorwärts
//NEG       Richtungssignal negativ / Transport rückwärts
//SET       Encoder auf Startwert setzten
//SETPOINT  Startwert Encoder
//r_mm_pro_Impuls  Auflösung Encoder mm pro Impuls
//
//[OUT]
//// mit den RP-Signalen kann direkt ein Ringpuffer angesteuert werden
//RP_POS    Richtungsimpuls positiv/vorwärts  (1 Zyklus)
//RP_NEG S  Richtungsimpuls negativ/rückwärts (1 Zyklus)
//ENCODER_mm  Encoder-Wert auf Auflösung umgerechnet [mm]
//
//[IN_OUT]
//tmpByte       Statisches Hilfsbyte (Merkerersatz)
//io_ENCODER   Positionswert des Encoders in Impulsen
//
//FC_ENO :  Richtungsimpuls vorwärts oder Richtungsimpuls rückwärts
//
//AUTOR: Stefan Maag, Dipl.-Ing. (FH) Elektrotechnik
//DATUM: 9/2004
//
//AENDERUNGSVERMERKE:
//--------------------------------------------------------------------------------
//DATUM        NAME    AENDERUNG
//--------------------------------------------------------------------------------
//29.07.2008  S.Maag   OUT_ENCODER als DINT
//                     Richtungsimpule für vw/rw (RP_VW / RP_RW) hinzugefügt
//                     FC_ENO = RP_POS oder RP_NEG
//
//21.10.2014  S.Maag   Ausgang ENCDER_mm und Eingang r_mm_pro_Impuls
//                     Umrechnung Encoderwert auf mm, dadurch Vereinfachung
//                     des Folgeprogramms => einzelne Umrechungen entfallen
//
//--------------------------------------------------------------------------------
//
//HINWEISE:
AUTHOR : 'S.Maag'
FAMILY : Maagic7
VERSION : 2.0


VAR_INPUT
  SENSOR : BOOL ;	//Eingang Encodersignal
  POS : BOOL ;	//Richtungssignal positiv / vorwärts
  NEG : BOOL ;	//Richtungssignal negativ / rückwärts
  SET : BOOL ;	//EncoderWert auf SetPoint
  SETPOINT : DINT ;	//ENCODER Wert SetPoint
  r_mm_pro_Impuls : REAL ;	//Auflösung mm pro Impuls
END_VAR
VAR_OUTPUT
  RP_POS : BOOL ;	//RichtungsImpuls positiv/vorwärts (Flanke f. Ringpuffer)
  RP_NEG : BOOL ;	//RichtungsImpuls negativ/rückwärts (Flanke f. Ringpuffer)
  ENCODER_mm : DINT ;	//Encoder umgerechnet auf mm Auflösung
END_VAR
VAR_IN_OUT
  memByte : BYTE ;	//Hilfsbyte
  io_ENCODER_IMP : DINT ;	//EncoderWert [Impulse]
END_VAR
VAR_TEMP
  tmpFP : BOOL ;	//positive Flanke Sensor Encoder
  tmpFN : BOOL ;	//negative Flanke Sensor Encoder
  tmpBit2 : BOOL ;
  tmpBit3 : BOOL ;
  tmpBit4 : BOOL ;
  tmpBit5 : BOOL ;
  tmpBit6 : BOOL ;
  tmpBit7 : BOOL ;
  FLK_NEG : BOOL ;
  FLK_POS : BOOL ;
  tmp_dResult : DINT ;
  tmp_dVAL : DINT ;
  tmp_rKomma : REAL ;
  tmp_ENCODER_LO : DWORD ;
  tmp_ENCODER_HI : DWORD ;
END_VAR
BEGIN
NETWORK
TITLE =Hilfsbyte in Lokaldatenbereich kopieren

      L     #memByte;
      T     LB     0;
NETWORK
TITLE =Flankenauswertung Sensor

      U     #SENSOR;
      FP    #tmpFP;
      =     #FLK_POS;

      U     #SENSOR;
      FN    #tmpFN;
      =     #FLK_NEG;
NETWORK
TITLE =Richtungsimpulse mit definiertem Wert (LOW) vorbelegen

      CLR   ;
      =     #RP_POS;
      =     #RP_NEG;

NETWORK
TITLE =SET: Encoder auf Startwert stellen

      U     #SET;
      SPBNB _001;
      L     #SETPOINT;
      T     #io_ENCODER_IMP;
_001: NOP   0;
NETWORK
TITLE =Encoder-Wert bei Flanke und Richtungssignal weiterzählen

      U     #FLK_POS; // Pos. Flanke Encoder
      U     #POS; // Ansteuersignal positiv
      SPB   pos; // zähle positiv / vorwärts
      U     #FLK_NEG; // Neg. Flanke Encoder
      U     #NEG; // Ansteuersignal negativ
      SPB   neg; // zähle negativ / rückwärts
      CLR   ;
      SAVE  ;
      SPA   END;

pos:  SAVE  ; // FC_ENO = HIGH
      =     #RP_POS; // Richtungsimpuls positiv/vw.
      L     #io_ENCODER_IMP;
      +     L#1;
      T     #io_ENCODER_IMP;
      SPA   END;

neg:  SAVE  ; // FC_ENO = HIGH
      =     #RP_NEG; // Richtungsimpuls negativ/rw.
      L     #io_ENCODER_IMP;
      +     L#-1;
      T     #io_ENCODER_IMP;

NETWORK
TITLE =Hilfsbyte wieder zurück kopieren und Encoder mm berechnen

END:  L     #io_ENCODER_IMP;
      DTR   ;
      L     #r_mm_pro_Impuls;
      *R    ;
      RND   ;
      T     #ENCODER_mm;

      L     LB     0;
      T     #memByte;

      BEA   ;
NETWORK
TITLE =
//18.10.2016 S.Maag
//Ansatz für korrekte Berechnung bei grossen Zahlen.
//Da REAL nur mit 23 Bit Genauigkeit arbeitet, wird automatisch
//gerundet, was zu fatalen Fehlern führt, wenn Wegdifferenzen berechnet werden
//sollen.
//
//FUNKTIONIERT NOCH NICHT: Siehe FC83 für korrekte Berechnung
// 1. ganzahlige mm Encoderwert berechnen

      L     #r_mm_pro_Impuls; // mm pro Impulse  [REAL]
      TRUNC ; // nach DINT : Kommastellen abgeschnitten
      T     #tmp_dVAL; // Wert vor Komma DINT (ganzzahlige mm Aufloesung)
      L     #io_ENCODER_IMP; // ENCODER_IMP
      *D    ; // *D := ganzahlige mm Encoder
      T     #tmp_dResult; // Zwischenergebnis := Encoderwert ganzahlige mm

// 2. Nachkommawert Aufloesung Encoder mm
      L     #r_mm_pro_Impuls; // mm pro Impulse  [REAL]
      L     #tmp_dVAL;
      DTR   ;
      -D    ;
      T     #tmp_rKomma; // r_mm_pro_Impulse : Wert nach Kommastelle

// 3. Encoder Impulse 32 Bit in 2 Berechnungen zerlegen 16x HiBit + 16x LoBit
      L     #io_ENCODER_IMP;
      UD    DW#16#FFFF0000;
      T     #tmp_ENCODER_HI; // ENCODER Hi zwischenspeichern
      DTR   ;
      L     #tmp_rKomma;
      *R    ;
      RND   ;
      L     #tmp_dResult;
      +D    ;
      T     #tmp_dResult; // Zwischenergebnis

      L     #io_ENCODER_IMP;
      L     #tmp_ENCODER_HI;
      -D    ;
      T     #tmp_ENCODER_LO;
      DTR   ;
      L     #tmp_rKomma;
      *R    ;
      RND   ;
      L     #tmp_dResult;
      +D    ;
      T     #tmp_dResult; // Zwischenergebnis



END_FUNCTION

FUNCTION "m7b_L_MESS" : VOID
TITLE =Längenmessung mit Lichtschranke und Encoder
//
//AUTOR: Stefan Maag, Dipl.-Ing. (FH) Elektrotechnik
//DATUM: 8/2008
//
//AENDERUNGSVERMERKE:
//--------------------------------------------------------------------------------
//DATUM        NAME    AENDERUNG
//--------------------------------------------------------------------------------
//
//--------------------------------------------------------------------------------
//
//HINWEISE:
AUTHOR : 'S.Maag'
FAMILY : Maagic7
VERSION : 0.1


VAR_INPUT
  LS : BOOL ;	//Lichtschranke
  ENCODER : DINT ;	//Wegwert ENCODER
END_VAR
VAR_OUTPUT
  IST : DINT ;
END_VAR
VAR_IN_OUT
  memByte : BYTE ;	//Hilfsbyte
  memWEG : DINT ;
END_VAR
VAR_TEMP
  tmpFP : BOOL ;	//positive Flanke Sensor Encoder
  tmpFN : BOOL ;	//negative Flanke Sensor Encoder
  tmpBit2 : BOOL ;
  tmpBit3 : BOOL ;
  tmpBit4 : BOOL ;
  tmpBit5 : BOOL ;
  tmpBit6 : BOOL ;
  tmpBit7 : BOOL ;
  FLK_POS : BOOL ;
  FLK_NEG : BOOL ;
END_VAR
BEGIN
NETWORK
TITLE =Hilfsbyte in Lokaldatenbereich kopieren

      L     #memByte;
      T     LB     0;

NETWORK
TITLE =Wegwert Encoder bei Lichtschranke belegt speichern

      U     #LS;
      FP    #tmpFP;
      SPBNB _001;
      L     #ENCODER;
      T     #memWEG;
      SET   ;
      SAVE  ;
      CLR   ;
_001: U     BIE;
      =     #FLK_POS;
NETWORK
TITLE =Negative Flanke als FC-ENO Ausgang speichern
//Mit der negativen Flanke am ENO-Ausgang kann bei Messende z.B. der aktuelle
//Messert umkopiert werden
      U     #LS;
      FN    #tmpFN;
      =     #FLK_NEG;
      SAVE  ;
NETWORK
TITLE =Messung läuft? Messwert ermitteln! bzw. letzten Wert ausgeben

      O     #LS; // Wenn Lichtschranke belegt, dann messen
      O     #FLK_NEG; // auch bei neg. Flanke nochmal bearbeiten, dies ist
      SPB   DO; // nötig, da dann der Istwert in tmpWeg gespeichert werden muss

      L     #memWEG; // Hilfsspeicher Weg als Ist ausgeben
      T     #IST; // wenn Messung beendet ist
      SPA   END;

NETWORK
TITLE =Aktuellen Istwert des Wegs berechnen
//Weg berechnen, den Lichtschranke belegt ist.
//Um den Istwert konsistent zu halten wird bei negativer Flanke des LS der
//Istwert in memWeg gespeichert und dann ständig ausgegeben. Dies ist nötig, da
//ein FC die Ausgänge selbst nichgt konsistent halten kann.
DO:   L     #ENCODER; // Wert vom Encoder
      L     #memWEG; // gespeicherter Wert bei LS belegt
      UC    "m7a_ABS_DIFF_DINT"; // absolute Differenz
      T     #IST; // aktueller Istwert Länge

      UN    #FLK_NEG; // Bei negativer Flanke der Lichtschranke
      SPB   END; // den Istwert als tmpWeg speichern. Dieser wird dann
      T     #memWEG; // ständig als IST ausgegeben, wenn LS nicht belegt ist.
NETWORK
TITLE =Hilfsbyte wieder zurück kopieren

END:  L     LB     0;
      T     #memByte;

END_FUNCTION

FUNCTION "m7b_STATUS_MOTOR" : VOID
TITLE =Motorstatus für OP erzeugen
//AUTOR: Stefan Maag, Dipl.-Ing. (FH) Elektrotechnik
//DATUM: 03/2005
//INTERNET: www.maagic7.de
//
//AENDERUNGSVERMERKE:
//--------------------------------------------------------------------------------
//DATUM        NAME            AENDERUNG
//--------------------------------------------------------------------------------
//
//--------------------------------------------------------------------------------
//
//HINWEISE:
AUTHOR : 'S.Maag'
FAMILY : Maagic7
VERSION : 0.1


VAR_INPUT
  VW : BOOL ;	//vorwärts EIN
  RW : BOOL ;	//rückwärts EIN
  ERR : BOOL ;	//Signal Störung
END_VAR
VAR_OUTPUT
  STATUS : INT ;
END_VAR
BEGIN
NETWORK
TITLE =
//0 = aus
//1 = ein
//2 = Störung
//3 = links bzw. rückwärts
      L     2;
      U     #ERR;
      SPB   SAVE;

      L     3;
      U     #RW;
      SPB   SAVE;

      L     1;
      U     #VW;
      SPB   SAVE;
      L     0;

SAVE: T     #STATUS;

      O     #VW;
      O     #RW;
      SAVE  ;
      CLR   ;
END_FUNCTION

FUNCTION "m7b_STATUS_DRIVE_EX" : VOID
TITLE =EXTENDED DRIVE STAUTS
//
//AUTOR: Stefan Maag, Dipl.-Ing. (FH) Elektrotechnik
//DATUM: 12/2012
//INTERNET: www.maagic7.de
//
//AENDERUNGSVERMERKE:
//--------------------------------------------------------------------------------
//DATUM        NAME            AENDERUNG
//--------------------------------------------------------------------------------
//
//--------------------------------------------------------------------------------
//
//HINWEISE: Entstand aus FC81 STATUS_MOTOR
AUTHOR : 'S.Maag'
FAMILY : Maagic7
VERSION : 0.1


VAR_INPUT
  START_FWD : BOOL ;	//START forward
  START_REV : BOOL ;	//START reverse
  ERR : BOOL ;	//ERROR
  AUTO : BOOL ;	//Automatic
END_VAR
VAR_OUTPUT
  STATUS : INT ;
END_VAR
BEGIN
NETWORK
TITLE =



NETWORK
TITLE =
//0 = AUS
//1 = EIN
//2 = Störung
//3 = Rückw. (links)
//4 = HAND AUS
//5 = HAND EIN
//6 = HAND RW
      L     2;
      U     #ERR;
      SPB   SAVE;

      L     3;
      U     #AUTO;
      U     #START_REV;
      SPB   SAVE;

      L     1;
      U     #AUTO;
      U     #START_FWD;
      SPB   SAVE;

      L     6;
      UN    #AUTO;
      U     #START_REV;
      SPB   SAVE;

      L     5;
      UN    #AUTO;
      U     #START_FWD;
      SPB   SAVE;

      L     4;
      UN    #AUTO;
      UN    #START_FWD;
      UN    #START_REV;
      SPB   SAVE;

      L     0;

SAVE: T     #STATUS;

      O     #START_FWD;
      O     #START_REV;
      SAVE  ;
      CLR   ;
END_FUNCTION

FUNCTION "m7b_STATUS_VALVE" : VOID
TITLE =Detailed Valve Status
//Attention: Different STATUS values for AUTO and HAND mode possible.
//in Hand Mode 10 is added to the STATUS value. This is to draw the HMI-Valve
//with a different frame color in HAND Mode.
//Generally I use orange to indicate HAND Mode.
//
//If different color for Hand Mode should be deactivated, call
//the FC with AUTO=TRUE!
//
//AUTOR: Stefan Maag, Dipl.-Ing. (FH) Elektrotechnik
//DATUM: 9/2018
//
//AENDERUNGSVERMERKE:
//--------------------------------------------------------------------------------
//DATUM        NAME        AENDERUNG
//--------------------------------------------------------------------------------
//
//--------------------------------------------------------------------------------
//
//HINWEISE:
AUTHOR : 'S.Maag'
FAMILY : Maagic7
VERSION : 0.1


VAR_INPUT
  COIL_A : BOOL ;	//Coil A activated (working position / open)
  COIL_B : BOOL ;	//Coil B activated (home position / close)
  POS_A : BOOL ;	//Position A reached (working position / open)
  POS_B : BOOL ;	//Position B reached (home position / closed)
  ERR_POS_A : BOOL ;	//Error Position A (working position / open)
  ERR_POS_B : BOOL ;	//Error Position B (home position / closed)
  AUTO : BOOL ;	//Auto Mode (If NOT AUTO THEN ADD (STATUS, 10)) for different Frame color in HAND
END_VAR
VAR_OUTPUT
  STATUS : INT ;
END_VAR
BEGIN
NETWORK
TITLE =



NETWORK
TITLE =Statusanzeige bearbeiten
//AUTO : HAND
//0    : 10    = no Action / keine Aktion aktiv bzw. undefiniert
//1    : 11    = Position A (working position / 'open')
//2    : 12    = Position B (homne psotion / 'closed')
//3    : 13    = moving to A
//4    : 14    = moving to B
//5    : 15    = Error Position A
//6    : 16    = Error Position B
      L     5; // Fehler Position A (Arbeitsstellung)
      U     #ERR_POS_A;
      SPB   SAVE;

      L     6; // Fehler Position B (Grundstellung)
      U     #ERR_POS_B;
      SPB   SAVE;

      L     1; // Position A erreicht (Arbeitsstellung)
      U     #POS_A;
      UN    #COIL_B;
      SPB   SAVE;

      L     2; //  Position B erreicht (Grundstellung)
      U     #POS_B;
      UN    #COIL_A;
      SPB   SAVE;

      L     3; // fährt zu Position A (Arbeitsstellung)
      U     #COIL_A;
      SPB   SAVE;

      L     4; // fährt zu Position B (Grundstellung)
      U     #COIL_B;
      SPB   SAVE;

      L     0;

SAVE: T     #STATUS;

NETWORK
TITLE =IF NOT AUTO THEN ADD(STATUS, 10)
//ADD 10 to STATUS in Manual Mode
//This is used to draw the HMI-Valve in a different frame color in HAND Mode.
//Generally I use orange to indicate HAND Mode
      UN    #AUTO;
      SPBNB _001;
      L     #STATUS;
      L     10;
      +I    ;
      T     #STATUS;
_001: NOP   0;
NETWORK
TITLE =

      SET   ;
      SAVE  ;
      CLR   ;

END_FUNCTION

FUNCTION "m7b_NiveauSchalter_REAL" : VOID
TITLE =Niveau-Schalter mit Min/Max Hysterese, Min- oder Max- schaltend
//Niveau-Schalter mit Min/Max Hysterese, Min- oder Max- schaltend
//
//Das Schaltsignal kann über das I/O-Bit OUT und am FC-ENO-Ausgang abgenommen
//werden. Somit kann der FC direkt in logischen Verknüpfungen verschaltet werden.
//
//VERWENDUNG:
//2-Punkt-Regler
//Befüllen oder entleeren von Tanks mit Füllstandsmesser
//Heizen bzw. kühlen
//
//VALUE : Istwert (Temperatur, Druck, Füllstand ...)
//MIN   : Minimalwert (Ein bei Min-schaltend bzw. Aus bei Max-schaltend)
//MAX   : Maximalwert (Aus bei Min-schaltend bzw. Ein bei Max-schaltend)
//
//Fkt_Min_Max:
//  0 = Minimumschaltend
//      Beim Minimum wird eingeschaltet bis das Maximum erreicht ist, dann aus
//      (z.B. befüllen, heizen)
//
//  1 = Maximumschaltend
//      Beim Maximu wird eingeschaltet bis das Minimum erreicht ist, dann aus
//      (z.B. entleeren, kühlen)
//
//OUT : Schaltsignal
//
//AUTOR: Stefan Maag, Dipl.-Ing. (FH) Elektrotechnik
//DATUM: 7/2004
//INTERNET: www.maagic7.de
//
//AENDERUNGSVERMERKE:
//--------------------------------------------------------------------------------
//DATUM        NAME            AENDERUNG
//--------------------------------------------------------------------------------
//
//--------------------------------------------------------------------------------
//
//HINWEISE:
AUTHOR : 'S.Maag'
FAMILY : Maagic7
VERSION : 0.1


VAR_INPUT
  VALUE : REAL ;	//Istwert
  MIN : REAL ;	//Minimalwert Hysterese
  MAX : REAL ;	//Maximalwert Hysterese
  cfg_Min_Max : BOOL ;	//0=MinSchaltend (z.B. befüllen, heizen) 1=MaxSchaltend (z.B. entleeren, kühlen)
END_VAR
VAR_IN_OUT
  OUT : BOOL ;	//Hilfsbit, Hilfmerker
END_VAR
BEGIN
NETWORK
TITLE =
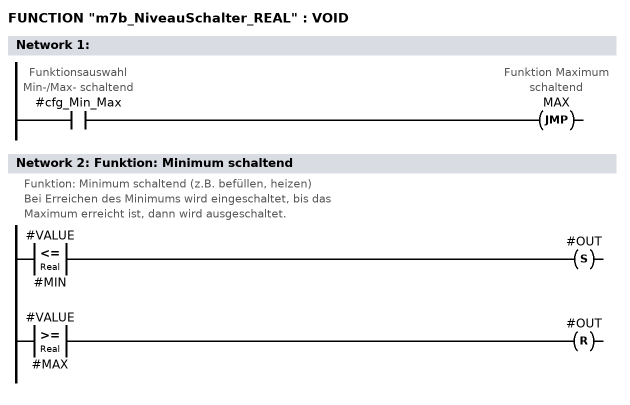

      U     #cfg_Min_Max; // Funktionsauswahl Min-/Max- schaltend
      SPB   MAX; // Funktion Maximum schaltend

NETWORK
TITLE =Funktion: Minimum schaltend
//Funktion: Minimum schaltend (z.B. befüllen, heizen)
//Bei Erreichen des Minimums wird eingeschaltet, bis das
//Maximum erreicht ist, dann wird ausgeschaltet.
      U(    ;
      L     #VALUE;
      L     #MIN;
      <=R   ;
      )     ;
      S     #OUT;
      U(    ;
      L     #VALUE;
      L     #MAX;
      >=R   ;
      )     ;
      R     #OUT;
      NOP   0;
NETWORK
TITLE =

      SPA   END;
MAX:  NOP   0;
NETWORK
TITLE =Funktion: Maximum schaltend
//Funktion: Maximum schaltend (z.B. entleeren, kühlen)
//Bei Erreichen des Maximus wird eingeschaltet, bis das
//Minimum wieder erreicht ist, dann wird ausgeschaltet.
      U(    ;
      L     #VALUE;
      L     #MAX;
      >=R   ;
      )     ;
      S     #OUT;
      U(    ;
      L     #VALUE;
      L     #MIN;
      <=R   ;
      )     ;
      R     #OUT;
      NOP   0;
NETWORK
TITLE =Schaltsignal auf FC-ENO-Ausgang für direkte Weiterverschaltung

END:  U     #OUT;
      SAVE  ;
      CLR   ;

END_FUNCTION

FUNCTION "m7b_NiveauSchalter_INT" : VOID
TITLE =Niveau-Schalter mit Min/Max Hysterese, Min- oder Max- schaltend
//Niveau-Schalter mit Min/Max Hysterese, Min- oder Max- schaltend
//
//Das Schaltsignal kann über das I/O-Bit OUT und am FC-ENO-Ausgang abgenommen
//werden. Somit kann der FC direkt in logischen Verknüpfungen verschaltet werden.
//
//VERWENDUNG:
//2-Punkt-Regler
//Befüllen oder entleeren von Tanks mit Füllstandsmesser
//Heizen bzw. kühlen
//
//VALUE : Istwert (Temperatur, Druck, Füllstand ...)
//MIN   : Minimalwert (Ein bei Min-schaltend bzw. Aus bei Max-schaltend)
//MAX   : Maximalwert (Aus bei Min-schaltend bzw. Ein bei Max-schaltend)
//
//Fkt_Min_Max:
//  0 = Minimumschaltend
//      Beim Minimum wird eingeschaltet bis das Maximum erreicht ist, dann aus
//      (z.B. befüllen, heizen)
//
//  1 = Maximumschaltend
//      Beim Maximu wird eingeschaltet bis das Minimum erreicht ist, dann aus
//      (z.B. entleeren, kühlen)
//
//OUT : Schaltsignal
//
//AUTOR: Stefan Maag, Dipl.-Ing. (FH) Elektrotechnik
//DATUM: 7/2004
//INTERNET: www.maagic7.de
//
//AENDERUNGSVERMERKE:
//--------------------------------------------------------------------------------
//DATUM        NAME            AENDERUNG
//--------------------------------------------------------------------------------
//
//--------------------------------------------------------------------------------
//
//HINWEISE:
AUTHOR : 'S.Maag'
FAMILY : Maagic7
VERSION : 0.1


VAR_INPUT
  VALUE : INT ;	//Istwert
  MIN : INT ;	//Minimalwert Hysterese
  MAX : INT ;	//Maximalwert Hysterese
  cf_Min_Max : BOOL ;	//0=MinSchaltend (z.B. befüllen, heizen) 1=MaxSchaltend (z.B. entleeren, kühlen)
END_VAR
VAR_IN_OUT
  OUT : BOOL ;	//Hilfsbit, Hilfmerker
END_VAR
BEGIN
NETWORK
TITLE =
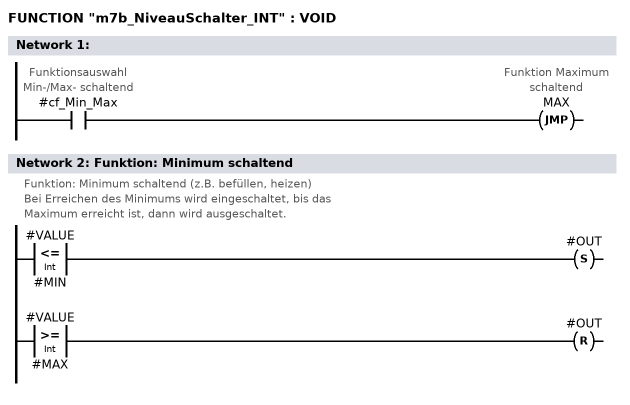

      U     #cf_Min_Max; // Funktionsauswahl Min-/Max- schaltend
      SPB   MAX; // Funktion Maximum schaltend

NETWORK
TITLE =Funktion: Minimum schaltend
//Funktion: Minimum schaltend (z.B. befüllen, heizen)
//Bei Erreichen des Minimums wird eingeschaltet, bis das
//Maximum erreicht ist, dann wird ausgeschaltet.
      U(    ;
      L     #VALUE;
      L     #MIN;
      <=I   ;
      )     ;
      S     #OUT;
      U(    ;
      L     #VALUE;
      L     #MAX;
      >=I   ;
      )     ;
      R     #OUT;
      NOP   0;
NETWORK
TITLE =

      SPA   END;
MAX:  NOP   0;
NETWORK
TITLE =Funktion: Maximum schaltend
//Funktion: Maximum schaltend (z.B. entleeren, kühlen)
//Bei Erreichen des Maximus wird eingeschaltet, bis das
//Minimum wieder erreicht ist, dann wird ausgeschaltet.
      U(    ;
      L     #VALUE;
      L     #MAX;
      >=I   ;
      )     ;
      S     #OUT;
      U(    ;
      L     #VALUE;
      L     #MIN;
      <=I   ;
      )     ;
      R     #OUT;
      NOP   0;
NETWORK
TITLE =Schaltsignal auf FC-ENO-Ausgang für direkte Weiterverschaltung

END:  U     #OUT;
      SAVE  ;
      CLR   ;

END_FUNCTION

FUNCTION "m7b_OFF_HAND_AUTO" : VOID
TITLE =Standardfunktion zur Betriebsartenumschaltung OFF/HAND/AUTO
//Betriebsartenumschaltung AUS/HAND/AUTO mit TriState Schaltfunktion
//Es kann wahlweise über OFF, SET_HAND und SET_AUTO oder einen Softwareschalter
//vom OP/PC geschaltet werden. Alle Schaltfunktionen sind parallel anwendbar. Bei
//einer Schaltstellungsänderung wird der Softwareschalter automatisch angepaßt.
//
//Verwendung: Konsistente Betriebsartenumschaltung AUS/HAND/OFF von
//            HMI (Softwareschalter) und Vor-Ort-Tasten
//
//Hinweis   : OFF hat die höchste priorität, dann Hand, dann AUTO
//            Die Binäreingänge haben Vorrang vor dem Softwareschalter.
//            Werden die Binäreingänge nicht benötigt, dann mit FALSE
//            beschalten.
//
//[IN]
//OFF       : Hi an diesem Eingang Schaltet auf AUS - höchste Priotiätät
//SET_MAN   : Schaltet um auf den Zustand 1: HAND=1, AUTO=0
//SET_AUTO  : Schaltet um auf den Zustand 2: HAND=0, AUTO=1
//
//FRG_AUTO  : Automatik erlauben: Bei Übergang 1->0 wird auf AUS geschaltet
//FRG_SOFT  : Freigabe für Softwareschalter. Bei Lo wird der Softwareschalter
//            gesperrt. Es wird nur die Umschaltfunktion des Softwareschalters
//            gesperrt. Die aktuelle Schaltstellung wird weiterhin angezeigt.
//
//[IN_OUT]
//S_SOFT    : Softwareschalter im INT-Format 0:=AUS; 1:=HAND; 2:=AUTO;
//memByte   : statosches Hilfbyte für Zustandsspeicherung
//
//S_SOFT    : Softwareschalter 0/1/2 eines Softwareschalter,
//            z.B. von OP, Visualisierung
//            0 : Hand=0, Auto=0
//            1 : Hand=1, Auto=0
//            2 : Hand=0, Auto=1
//[OUT]
//HAND      : Ausgang Schaltzustand HAND
//AUTO      : Ausgang Schaltzustand AUTO
//
//FC.ENO    : Ausgang ist 1, wenn ein Ereignis OFF/HAND/AUTO auftritt,
//            dass durch den Softwareschalter ausglöst wurde (=HMI/USER-action)
//
//AUTOR: Stefan Maag, Dipl.-Ing. (FH) Elektrotechnik
//SOURCE: basiert auf Kombination von FC48 'TriStateSwitch' und FC45 'Hand/Auto'
//DATUM: 06/2012
//INTERNET: www.maagic7.de
//
//AENDERUNGSVERMERKE:
//--------------------------------------------------------------------------------
//DATUM        NAME      AENDERUNG
//--------------------------------------------------------------------------------
//03.09.2018   S.Maag    FRG_AUTO hinzugefügt/übernommen (war schon länger bei
//                       Maschinen verwendet, welche global USER_MODE_CONTROL
//                       hatten.)
//                       FC.ENO := SoftwareSwitch/HMI/USER-Action
//--------------------------------------------------------------------------------
//
//HINWEISE:
AUTHOR : 'S.Maag'
FAMILY : Maagic7
VERSION : 1.0


VAR_INPUT
  OFF : BOOL ;	//Eingang für Ausschalter
  SET_HAND : BOOL ;	//Eingang für Zustand 1 (Hand) einschalten
  SET_AUTO : BOOL ;	//Eingang für Zustand 2 (Auto) einschalten
  FRG_AUTO : BOOL ;	//Automatikbetrieb erlauben: Bei Übergang 1->0 wird auf AUS geschaltet
  FRG_SOFT : BOOL ;	//Freigabe für Softwareschalter
END_VAR
VAR_OUTPUT
  HAND : BOOL ;	//HAND
  AUTO : BOOL ;	//AUTO
  EVT_OFF : BOOL ;	//Event: Mode OFF activated
  EVT_HAND : BOOL ;	//Event: Mode HAND activated
  EVT_AUTO : BOOL ;	//Event: Mode AUTO activated
  DSP_MODE : INT ;	//Display actual mode: 0:=OfF; 1:=HAND; 2:=AUTO
END_VAR
VAR_IN_OUT
  S_SOFT : INT ;	//Softwareschalter
  memByte : BYTE ;	//statischer Hiflsspeicher
END_VAR
VAR_TEMP
  lb_HAND : BOOL ;	//STATIC BYTE: Output HAND
  lb_AUTO : BOOL ;	//STATIC BYTE: Output AUTO
  lb_2 : BOOL ;	//STATIC BYTE:
  lb_LAST_STATE_AUTO : BOOL ;	//STATIC BYTE: last state was AUTO
  lb_EVT_OFF : BOOL ;	//STATIC BYTE: Event OFF
  lb_EVT_HAND : BOOL ;	//STATIC BYTE: Event HAND
  lb_EVT_AUTO : BOOL ;	//STATIC BYTE: Event AUTO
  lb_HM_FN_FRG_AUTO : BOOL ;	//STATIC BYTE: FTrig FRG_AUTO
  SOFT_STATE_HAND : BOOL ;	//Software Switch is in position HAND
  SOFT_STATE_AUTO : BOOL ;	//Software Switch is in position AUTO
  evt_FRG_OFF : BOOL ;	//Event AUTO-ENABLE OFF
  MSG_S_SOFT_ACTION : BOOL ;	//Software Switch action (HMI/User Operation)
END_VAR
BEGIN
NETWORK
TITLE =Dauerhaften Zwischenspeicher in Lokaldatenbereich
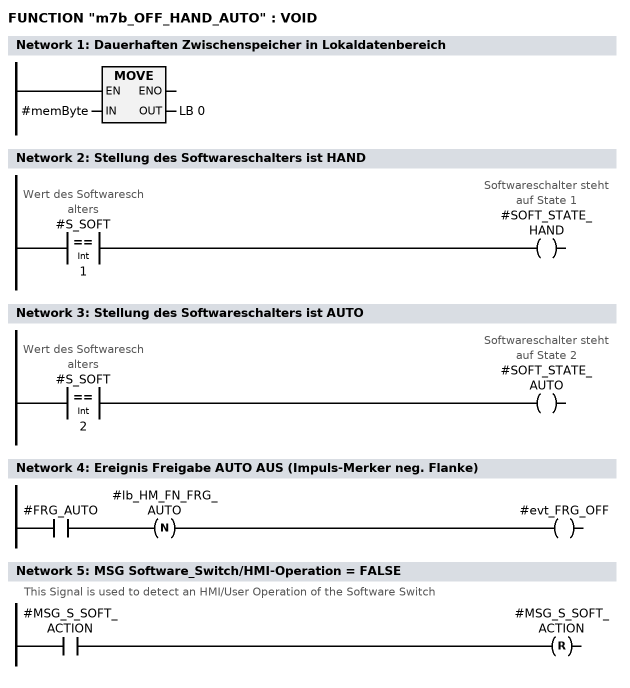

      L     #memByte;
      T     LB     0;
      NOP   0;
NETWORK
TITLE =Stellung des Softwareschalters ist HAND

      L     #S_SOFT; // Wert des Softwareschalters
      L     1;
      ==I   ;
      =     #SOFT_STATE_HAND; // Softwareschalter steht auf State 1

NETWORK
TITLE =Stellung des Softwareschalters ist AUTO

      L     #S_SOFT; // Wert des Softwareschalters
      L     2;
      ==I   ;
      =     #SOFT_STATE_AUTO; // Softwareschalter steht auf State 2

NETWORK
TITLE =Ereignis Freigabe AUTO AUS (Impuls-Merker neg. Flanke)

      U     #FRG_AUTO;
      FN    #lb_HM_FN_FRG_AUTO;
      =     #evt_FRG_OFF;

NETWORK
TITLE =MSG Software_Switch/HMI-Operation = FALSE
//This Signal is used to detect an HMI/User Operation of the Software Switch
      U     #MSG_S_SOFT_ACTION;
      R     #MSG_S_SOFT_ACTION;
NETWORK
TITLE =Auswertung der verschiedenen Schaltfunktionen

      U     #OFF; // Eingang für OFF hat immer Vorrang
      SPB   OFF;

      U     #SET_HAND; // wenn beide Zustände gleichzeitig
      U     #SET_AUTO; // gesetzt werden sollen, dann OFF
      SPB   OFF;

      U     #SET_HAND; // Eingang Zustand 1 (HAND) setzen
      SPB   HAND; // Zustand 1 (HAND)

      U     #lb_AUTO; // Auto aktiv
      U     #evt_FRG_OFF; // neg. Flanke FRG_AUTO (evt. Freigabe AUS)
      SPB   OFF;

      U     #SET_AUTO; // Eingang Zustand 2 (AUTO) setzen
      U     #FRG_AUTO;
      SPB   AUTO; // Zustand 2 (AUTO)

      UN    #FRG_SOFT; // Wenn keine Freigabe für den Softwareschalter,
      SPB   IST; // dann Istzustand in Softwareschalter schreiben

      UN    #lb_HAND; // Wenn Schaltausgang HAND=Lo
      U     #SOFT_STATE_HAND; // und Softwareschalter Zustand 1 (Hand) angewählt
      S     #MSG_S_SOFT_ACTION; // Softwareschalter Bedienung
      SPB   HAND; // dann Zustand 1 (HAND) aktivieren

      UN    #lb_AUTO; // Wenn Schaltausgang AUTO = Lo
      U     #SOFT_STATE_AUTO; // und Softwareschalter Zustand 2 (AUTO) angewählt
      U     #FRG_AUTO; // Freigabe für Automatikbetrieb
      S     #MSG_S_SOFT_ACTION; // Softwareschalter Bedienung
      SPB   AUTO; // dann Zustand 2 (AUTO) aktivieren

      UN    #SOFT_STATE_HAND; // Softwareschalter Zustand 1 nicht angewählt
      UN    #SOFT_STATE_AUTO; // Softwareschalter Zustand 2 nicht angewählt
      S     #MSG_S_SOFT_ACTION; // Softwareschalter Bedienung
      SPB   OFF; // dann OFF

      U     #SOFT_STATE_AUTO; // Softwareschalter Zustand 2 AUTO angewählt
      UN    #FRG_AUTO; // keine AUTO-Freigabe
      SPB   IST; // dann Softwareschalter auf IST Betriebszustand

      SPA   NE3;

HAND: S     #lb_HAND; // Schaltausgang 1 setzen
      R     #lb_AUTO; // Schaltausgang 2 löschen
      R     #lb_LAST_STATE_AUTO; // letzter aktiver Zustand war S2 löschen
      L     1; // Softwareschalter auf 1
      SPA   SAVE;

AUTO: R     #lb_HAND; // Schaltausgang 1 löschen
      S     #lb_AUTO; // Schaltausgang 2 setzen
      S     #lb_LAST_STATE_AUTO; // letzter aktiver Zustand war S2 (merken)
      L     2; // Softwareschalter auf 2
      SPA   SAVE;

OFF:  R     #lb_HAND; // Schaltausgang 1 löschen
      R     #lb_AUTO; // Schaltausgang 2 löschen
      L     0; // Softwareschalter auf 0
      SPA   SAVE;

IST:  L     1;
      U     #lb_HAND; // Ausgang 1 (HAND) ist aktiv: State 1
      SPB   SAVE;
      L     2;
      U     #lb_AUTO; // Ausgang 2 (AUTO) ist aktiv: State 2
      SPB   SAVE;
      L     0;

SAVE: T     #S_SOFT; // Softwareschalter schreiben
NE3:  NOP   0;
NETWORK
TITLE =FC-Ausgang 'HAND' & 'Ereignis HAND'

      U     #lb_HAND;
      =     #HAND;
      FP    #lb_EVT_HAND;
      =     #EVT_HAND;
NETWORK
TITLE =FC-Ausgang 'AUTO' & 'Ereignis AUTO'

      U     #lb_AUTO;
      =     #AUTO;
      FP    #lb_EVT_AUTO;
      =     #EVT_AUTO;
NETWORK
TITLE =FC-Ausgang 'Ereignis OFF'

      UN    #lb_HAND;
      UN    #lb_AUTO;
      FP    #lb_EVT_OFF;
      =     #EVT_OFF;

NETWORK
TITLE =Anzeigeausgang aktiver Modus: DSP_MODE
//0 := OFF
//1 := HAND
//2 := AUTO
      L     1;
      U     #lb_HAND; // Ausgang 1 (HAND) ist aktiv: State 1
      SPB   sav9;
      L     2;
      U     #lb_AUTO; // Ausgang 2 (AUTO) ist aktiv: State 2
      SPB   sav9;
      L     0;
sav9: T     #DSP_MODE; // Anzeigeausgang angewählter Modus

NETWORK
TITLE =Lokalen Speicher wieder in dauerhaften Zwischenspeicher

      L     LB     0;
      T     #memByte;
      NOP   0;
NETWORK
TITLE =FC.ENO = HMI/User-Action (Software swicht operated)

      U(    ;
      O     #EVT_OFF; // Ereignis AUS
      O     #EVT_HAND; // Ereignis HAND
      O     #EVT_AUTO; // Ereignis AUTO
      )     ;
      U     #MSG_S_SOFT_ACTION; // Softwareschalter Bedienung
      SAVE  ; // auf FC-ENO-Ausgang geben


END_FUNCTION

FUNCTION "m7b_NiveauSchalter_DINT" : VOID
TITLE =Niveau-Schalter mit Min/Max Hysterese, Min- oder Max- schaltend
//Niveau-Schalter mit Min/Max Hysterese, Min- oder Max- schaltend
//
//Das Schaltsignal kann über das I/O-Bit OUT und am FC-ENO-Ausgang abgenommen
//werden. Somit kann der FC direkt in logischen Verknüpfungen verschaltet werden.
//
//VERWENDUNG:
//2-Punkt-Regler
//Befüllen oder entleeren von Tanks mit Füllstandsmesser
//Heizen bzw. kühlen
//
//VALUE : Istwert (Temperatur, Druck, Füllstand ...)
//MIN   : Minimalwert (Ein bei Min-schaltend bzw. Aus bei Max-schaltend)
//MAX   : Maximalwert (Aus bei Min-schaltend bzw. Ein bei Max-schaltend)
//
//Fkt_Min_Max:
//  0 = Minimumschaltend
//      Beim Minimum wird eingeschaltet bis das Maximum erreicht ist, dann aus
//      (z.B. befüllen, heizen)
//
//  1 = Maximumschaltend
//      Beim Maximu wird eingeschaltet bis das Minimum erreicht ist, dann aus
//      (z.B. entleeren, kühlen)
//
//OUT : Schaltsignal
//
//AUTOR: Stefan Maag, Dipl.-Ing. (FH) Elektrotechnik
//DATUM: 10/2014
//INTERNET: www.maagic7.de
//
//AENDERUNGSVERMERKE:
//--------------------------------------------------------------------------------
//DATUM        NAME            AENDERUNG
//--------------------------------------------------------------------------------
//
//--------------------------------------------------------------------------------
//
//HINWEISE: entstand aus Niveau-Schalter INT
AUTHOR : 'S.Maag'
FAMILY : Maagic7
VERSION : 0.1


VAR_INPUT
  VALUE : DINT ;	//Istwert
  MIN : DINT ;	//Minimalwert Hysterese
  MAX : DINT ;	//Maximalwert Hysterese
  cf_Min_Max : BOOL ;	//0=MinSchaltend (z.B. befüllen, heizen) 1=MaxSchaltend (z.B. entleeren, kühlen)
END_VAR
VAR_IN_OUT
  OUT : BOOL ;	//Hilfsbit, Hilfmerker
END_VAR
BEGIN
NETWORK
TITLE =
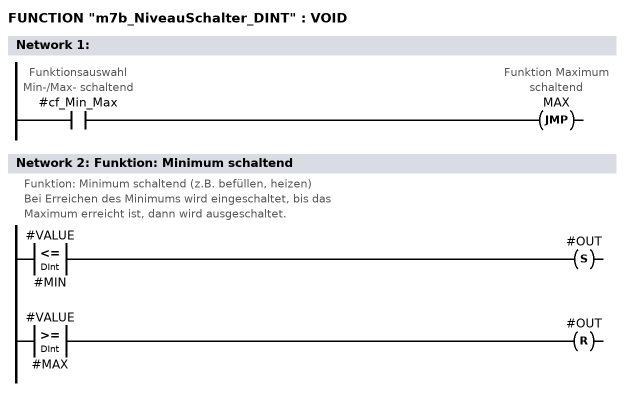

      U     #cf_Min_Max; // Funktionsauswahl Min-/Max- schaltend
      SPB   MAX; // Funktion Maximum schaltend

NETWORK
TITLE =Funktion: Minimum schaltend
//Funktion: Minimum schaltend (z.B. befüllen, heizen)
//Bei Erreichen des Minimums wird eingeschaltet, bis das
//Maximum erreicht ist, dann wird ausgeschaltet.
      U(    ;
      L     #VALUE;
      L     #MIN;
      <=D   ;
      )     ;
      S     #OUT;
      U(    ;
      L     #VALUE;
      L     #MAX;
      >=D   ;
      )     ;
      R     #OUT;
      NOP   0;
NETWORK
TITLE =

      SPA   END;
MAX:  NOP   0;
NETWORK
TITLE =Funktion: Maximum schaltend
//Funktion: Maximum schaltend (z.B. entleeren, kühlen)
//Bei Erreichen des Maximus wird eingeschaltet, bis das
//Minimum wieder erreicht ist, dann wird ausgeschaltet.
      U(    ;
      L     #VALUE;
      L     #MAX;
      >=D   ;
      )     ;
      S     #OUT;
      U(    ;
      L     #VALUE;
      L     #MIN;
      <=D   ;
      )     ;
      R     #OUT;
      NOP   0;
NETWORK
TITLE =Schaltsignal auf FC-ENO-Ausgang für direkte Weiterverschaltung

END:  U     #OUT;
      SAVE  ;
      CLR   ;

END_FUNCTION

FUNCTION "m7b_DRIVE_INFO" : VOID
TITLE =Drive Info
//Informationsfunktion für Antriebe:
//
//- Anzahl der Starts
//- Betriebsstunden
//- Service/Wartungsmeldung nach Anzahl der Starts und/oder Betriebsstunden
//- Service Warnmeldung Anzahl Starts oder Betriebstunden vor dem fälligen
//  Wartungstermin
//
//Mit Speicherung des Letzten Servicedatums sowie der Userkennung
//des Verantwortlichen
//
//PARAMETER IN:
//  SIGNAL:   Ansteuersignal des Antriebs (Antrieb Start)
//  SERVICE_RESET: Signal Service erledigt, Serviceintervall wird zurückgesetzt
//
//  DrvCfg: UDT91: UDT_SERVICE_CFG_DRV, Struktur mit Service Konfigurationsdaten
//
//PARAMETER IN_OUT:
//  DrvInf: UDT90: UDT_SERVICE_INF, Struktur in der Service- und Betriebsdaten
//
//                   gespeichert werden.
//
//AUTOR: Stefan Maag, Dipl.-Ing. (FH) Elektrotechnik
//DATUM: 5/2005
//
//AENDERUNGSVERMERKE:
//--------------------------------------------------------------------------------
//DATUM        NAME       AENDERUNG
//--------------------------------------------------------------------------------
//09.07.2017   S.Maag     Schon länger existierende Änderung mit RESET Button
//                        im udt_DrvInf in Bibliothek aufgenommen.
//                        Verleicherfehler im NW 9 für Starts Service behoben:
//                        war >=I statt >=D
//
//02.07.2012   S.Maag     Anzeige Rest- Zeit/Starts
//                        Vorbereitung UserName Service speichern
//--------------------------------------------------------------------------------
//
//HINWEISE:
AUTHOR : 'S.Maag'
FAMILY : Maagic7
VERSION : 0.1


VAR_INPUT
  SIGNAL : BOOL ;	//Motorsignal
  SERVICE_RESET : BOOL ;
  DrvCfg : "m7_udtServiceCFG_Drive";
END_VAR
VAR_OUTPUT
  SERVICE : BOOL ;	//Service fällig
  SERV_WARN : BOOL ;	//Service demnächst fällig
END_VAR
VAR_IN_OUT
  DrvInf : "m7_udtSericeInfo_Drive";
  HM : BOOL ;	//Hilfsmerker
END_VAR
VAR_TEMP
  DatumZeit : DATE_AND_TIME ;
  DATUM : DATE ;
  RET : INT ;
  SERVICE_H : BOOL ;
  SERVICE_STARTS : BOOL ;
  SERVICE_WARN_H : BOOL ;
  SERVICE_WARN_STARTS : BOOL ;
  RESET : BOOL ;
  tmpH : INT ;
END_VAR
BEGIN
NETWORK
TITLE =Anzahl der Starts zählen

      U     #SIGNAL;
      FP    #HM;
      SPBN  ne2;
      L     #DrvInf.STARTS; // Starts gesamt
      +     L#1;
      T     #DrvInf.STARTS;

      L     #DrvInf.SERVICE_STARTS; // Starts seit letzter Wartung
      +     L#1;
      T     #DrvInf.SERVICE_STARTS;

ne2:  NOP   0;

NETWORK
TITLE =(Betriebs-) Stunden zählen

      U     #SIGNAL; // Gerät eingeschaltet
      U     M    101.5; // Takt 1 Sekunde
      SPB   rcnt;
      SPA   ne3;

rcnt: L     #DrvInf.RUN_SEC; // Speicher für Sekunden
      +     1; // erhöhen
      T     #DrvInf.RUN_SEC;
      L     3600; // prüfen ob 1 Stunde vergangen = 3600 sec.
      >=I   ;
      SPB   rh; // wenn ja, Stunden bearbeiten
      SPA   ne3;

rh:   L     0; // neue Stunde: zuerst Sekunden löschen
      T     #DrvInf.RUN_SEC;

      L     #DrvInf.RUN_H; // Stundenspeicher erhöhen
      +     L#1;
      T     #DrvInf.RUN_H;
ne3:  NOP   0;
NETWORK
TITLE =(Betriebs-) Stunden seit letzter Wartung zählen

      U     #SIGNAL; // Gerät eingeschaltet
      U     M    101.5; // Takt 1 Sekunde
      SPB   scnt;
      SPA   ne4;

scnt: L     #DrvInf.SERVICE_SEC; // Speicher für Sekunden
      +     1; // erhöhen
      T     #DrvInf.SERVICE_SEC;
      L     3600; // prüfen ob 1 Stunde vergangen = 3600 sec.
      >=I   ;
      SPB   sh; // wenn ja, Stunden bearbeiten
      SPA   ne4;

sh:   L     0; // neue Stunde: zuerst Sekunden löschen
      T     #DrvInf.SERVICE_SEC;

      L     #DrvInf.SERVICE_H; // Stundenspeicher erhöhen
      +     L#1;
      T     #DrvInf.SERVICE_H;

ne4:  NOP   0;
NETWORK
TITLE =Resetbedingung
//RESET-Button über Service-Info-Struktur
//oder externer Eingang RESET
      O(    ;
      L     #DrvInf.RESET;
      L     1;
      ==I   ;
      )     ;
      O     #SERVICE_RESET;
      =     #RESET;
NETWORK
TITLE =Service Intervall rücksetzen

      UN    #RESET;
      SPB   ne5;
      L     L#0;
      T     #DrvInf.SERVICE_H;
      T     #DrvInf.SERVICE_SEC;
      T     #DrvInf.SERVICE_STARTS;

      CALL "READ_CLK" (// System Datum- und Uhrzeit
           RET_VAL                  := #RET,
           CDT                      := #DatumZeit);

      CALL "DT_DATE" (// Datum aus System Datum- Zeit lösen
           IN                       := #DatumZeit,
           RET_VAL                  := #DATUM);

      L     #DATUM;
      T     #DrvInf.LAST_SERVICE_DATE; // aktuelles Datum als letztes Servicedatum speichern

      L     0; // Reset-Befehl löschen
      T     #DrvInf.RESET;
ne5:  NOP   0;
NETWORK
TITLE =Anzeige Restzeit bis Service

      L     #DrvCfg.STD;
      L     #DrvInf.SERVICE_H;
      -I    ;
      SPPZ  sav1; // Springe wenn >=0
      L     0; // sonst auf 0 begrenzen
sav1: T     #DrvInf.DSP_SERVICE_H;
NETWORK
TITLE =Anzeige Reststarts bis Service

      L     #DrvCfg.STARTS;
      L     #DrvInf.SERVICE_STARTS;
      -D    ;
      SPPZ  sav2; // Springe wenn >=0
      L     L#0; // sonst auf 0 begrenzen
sav2: T     #DrvInf.DSP_SERVICE_STARTS;
NETWORK
TITLE =Betriebsstunden für Service prüfen
//Meldung Service ist jetzt fällig, nach Betriebsstunden
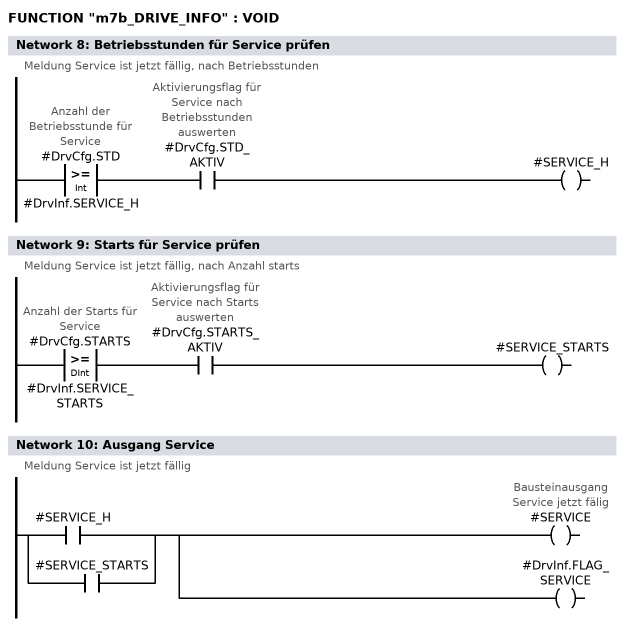
      U(    ;
      L     #DrvCfg.STD; // Anzahl der Betriebsstunde für Service
      L     #DrvInf.SERVICE_H; // Anzahl der Betriebsstunden seit letztem Service
      >=I   ;
      )     ;
      U     #DrvCfg.STD_AKTIV; // Aktivierungsflag für Service nach Betriebsstunden auswerten
      =     #SERVICE_H;

NETWORK
TITLE =Starts für Service prüfen
//Meldung Service ist jetzt fällig, nach Anzahl starts
      U(    ;
      L     #DrvCfg.STARTS; // Anzahl der Starts für Service
      L     #DrvInf.SERVICE_STARTS; // Anzahl der Starts seit letzem Servie
      >=D   ;
      )     ;
      U     #DrvCfg.STARTS_AKTIV; // Aktivierungsflag für Service nach Starts auswerten
      =     #SERVICE_STARTS;
NETWORK
TITLE =Ausgang Service
//Meldung Service ist jetzt fällig
      O     #SERVICE_H;
      O     #SERVICE_STARTS;
      =     #SERVICE; // Bausteinausgang Service jetzt fälig
      =     #DrvInf.FLAG_SERVICE;
NETWORK
TITLE =Betriebsstunden für Service Warnmeldung prüfen
//Warnung bzw- Hinweis, daß Service demnächst fällig ist, nach Betriebsstunden
      U(    ;
      L     #DrvCfg.STD;
      L     #DrvCfg.STD_DSP_MSG;
      -I    ;
      L     #DrvInf.SERVICE_H;
      >=I   ;
      )     ;
      U     #DrvCfg.STD_AKTIV; // Aktivierungsflag für Service nach Betriebsstunden auswerten
      =     #SERVICE_WARN_H;

NETWORK
TITLE =Starts für Service Warnmeldung prüfen
//Warnung bzw- Hinweis, daß Service demnächst fällig ist, nach Betriebsstunden
      U(    ;
      L     #DrvCfg.STARTS;
      L     #DrvCfg.STARTS_DSP_MSG;
      -D    ;
      L     #DrvInf.SERVICE_STARTS;
      >=D   ;
      )     ;
      U     #DrvCfg.STARTS_AKTIV; // Aktivierungsflag für Service nach Starts auswerten
      =     #SERVICE_WARN_STARTS;

NETWORK
TITLE =Ausgang Service demnächst

      O     #SERVICE_WARN_H;
      O     #SERVICE_WARN_STARTS;
      =     #SERV_WARN; // Bausteinausgang Service demnächst fällig
      =     #DrvInf.FLAG_SERVICE_WARN;
END_FUNCTION

FUNCTION "m7b_YK_INFO" : VOID
TITLE =Ventil/Schütz Info
//Informationsfunktion für Ventile/Schütze
//
//- Anzahl der Schaltungen
//- Service/Wartungsmeldung nach Anzahl der Schaltungen
//- Service Warnmeldung Anzahl Schaltungen vor dem fälligen Wartungstermin
//
//Mit Speicherung des Letzten Servicedatums sowie der Userkennung
//des Verantwortlichen
//
//PARAMETER IN:
//  SIGNAL:   Ansteuersignal des Antriebs (Antrieb Start)
//  SERVICE_RESET: Signal Service erledigt, Serviceintervall wird zurückgesetzt
//
//  YKCfg: UDT13: UDT_SERVICE_CFG_YK, Struktur mit Service Konfigurationsdaten
//
//PARAMETER IN_OUT:
//  YKInf: UDT12: UDT_SERVICE_INF, Struktur in der Service- und Betriebsdaten
//                 gespeichert werden.
//
//AUTOR: Stefan Maag, Dipl.-Ing. (FH) Elektrotechnik
//DATUM: 5/2005
//INTERNET: www.maagic7.de
//
//AENDERUNGSVERMERKE:
//--------------------------------------------------------------------------------
//DATUM        NAME        AENDERUNG
//--------------------------------------------------------------------------------
//
//--------------------------------------------------------------------------------
//
//HINWEISE:
AUTHOR : 'S.Maag'
FAMILY : Maagic7
VERSION : 0.1


VAR_INPUT
  SIGNAL : BOOL ;	//Motorsignal
  SERVICE_RESET : BOOL ;
  YKCfg : "m7_udt_ServiceCFG_YK";
END_VAR
VAR_OUTPUT
  SERVICE : BOOL ;	//Service fällig
  SERV_WARN : BOOL ;	//Service demnächst fällig
END_VAR
VAR_IN_OUT
  YKInf : "m7_udtServiceInfo_YK";
  HM : BOOL ;	//Hilfsmerker
END_VAR
VAR_TEMP
  DatumZeit : DATE_AND_TIME ;
  DATUM : DATE ;
  RET : INT ;
  SERVICE_SCHAKTUNGEN : BOOL ;
  SERVICE_WARN_SCHALTUNGEN : BOOL ;
END_VAR
BEGIN
NETWORK
TITLE =Anzahl der Starts zählen

      U     #SIGNAL;
      FP    #HM;
      SPBN  ne2;
      L     #YKInf.SCHALTUNGEN; // Starts gesamt
      +     L#1;
      T     #YKInf.SCHALTUNGEN;

      L     #YKInf.SERVICE_SCHALTUNGEN; // Starts seit letzter Wartung
      +     L#1;
      L     #YKInf.SERVICE_SCHALTUNGEN;

ne2:  NOP   0;

NETWORK
TITLE =Service Intervall rücksetzen

      UN    #SERVICE_RESET;
      SPB   ne5;
      L     L#0;
      T     #YKInf.SERVICE_SCHALTUNGEN;

      CALL "READ_CLK" (// System Datum- und Uhrzeit
           RET_VAL                  := #RET,
           CDT                      := #DatumZeit);
// Datum aus Systemzeit, Datum lösen
      CALL "DT_DATE" (
           IN                       := #DatumZeit,
           RET_VAL                  := #DATUM);

      L     #DATUM;
      T     #YKInf.LAST_SERVICE_DATE; // aktuelles Datum als letztes Servicedatum speichern
ne5:  NOP   0;
NETWORK
TITLE =Schaltungen für Service prüfen
//Meldung Service ist jetzt fällig, nach Anzahl Schaltungen
      U(    ;
      L     #YKCfg.SCHALTUNGEN; // Anzahl der Schaltungen für Service
      L     #YKInf.SERVICE_SCHALTUNGEN; // Anzahl der Schaltungen seit letzem Servie
      >=I   ;
      )     ;
      =     #SERVICE_SCHAKTUNGEN;
NETWORK
TITLE =Ausgang Service
//Meldung Service ist jetzt fällig
      O     #SERVICE_SCHAKTUNGEN;
      =     #SERVICE; // Bausteinausgang Service jetzt fälig
NETWORK
TITLE =Starts für Service Warnmeldung prüfen
//Warnung bzw- Hinweis, daß Service demnächst fällig ist, nach Betriebsstunden
      U(    ;
      L     #YKCfg.SCHALTUNGEN;
      L     #YKCfg.SCHALTUNGEN_DSP_MSG;
      -I    ;
      L     #YKInf.SERVICE_SCHALTUNGEN;
      >=I   ;
      )     ;
      =     #SERVICE_WARN_SCHALTUNGEN;
NETWORK
TITLE =Ausgang Service demnächst

      U     #SERVICE_WARN_SCHALTUNGEN;
      =     #SERV_WARN; // Bausteinausgang Service demnächst fällig

END_FUNCTION

FUNCTION "m7b_DAMPING_INT" : INT
TITLE =Kontinuierliche Mittelwertbildung eines INT-Wertes
//x   : neuer Mittelwert
//m   : letzter Mittelwert
//n   : Anzahl der Werte
//a   : Eingangswert
//
//x = m + (a-m)/n
//
//
//Bei jeder neuen Berechnung wird der FC-ENO Ausgang HIGH
//
//
//AUTOR: Stefan Maag, Dipl.-Ing. (FH) Elektrotechnik
//DATUM: 9/2005
//INTERNET: www.maagic7.de
//
//AENDERUNGSVERMERKE:
//--------------------------------------------------------------------------------
//DATUM        NAME            AENDERUNG
//--------------------------------------------------------------------------------
//
//--------------------------------------------------------------------------------
//
//HINWEISE:
AUTHOR : 'S.Maag'
FAMILY : Maagic7
VERSION : 2.0


VAR_INPUT
  IN_VALUE : INT ;	//Eingangswert
  IN_TAKT_RisingEdge : BOOL ;	//Taktflanke Zeittakt Dämpfung
  IN_rDampingFactor : REAL ;	//Dämpfungsfaktor muss >1 sein
END_VAR
VAR_IN_OUT
  IO_SENSOR_DAMP : REAL ;
END_VAR
VAR_TEMP
  rDamping : REAL ;
END_VAR
BEGIN
NETWORK
TITLE =

      SET   ;
      SAVE  ;
      CLR   ;

NETWORK
TITLE =Dämpfung des Sensorwertes
//Durch das aufaddieren eines Teils der Differenz zum aktuellen Analogwert
//läuft der gedämpfte Wert dem Analogwert immer etwas hinterher. Es ergibt sich
//ein exponentieller Nachlauf (vgl. Kondensator Ladekurve) bei einem
//Dämpfungsfaktor von 2 erhält man nach 5 Impulsen ca. 96.9%, nach 7 Impulsen ca.
//99.2% Sensorwertes. Je höher der Dämpfungsfaktor, desto langsamer läuft der
//Wert hinterher.
      UN    #IN_TAKT_RisingEdge;
      SPB   end;

      L     #IN_rDampingFactor; // sicherstellen, dass
      L     1.000000e+000; // Dämpfungsfaktor >=1.0
      <R    ;
      SPB   sav;
      TAK   ;
sav:  T     #rDamping;
      L     #IN_VALUE;
      ITD   ;
      DTR   ;
      L     #IO_SENSOR_DAMP;
      -R    ;
      L     #rDamping;
      /R    ;
      L     #IO_SENSOR_DAMP;
      +R    ;
      T     #IO_SENSOR_DAMP;
end:  L     #IO_SENSOR_DAMP;
      RND   ;
      T     #RET_VAL;
END_FUNCTION

FUNCTION "m7b_CONT_MITTEL_DINT" : VOID
TITLE =Kontinuierliche Mittelwertbildung eines DINT-Wertes
//x   : neuer Mittelwert
//m   : letzter Mittelwert
//n   : Anzahl der Werte
//a   : Eingangswert
//
//x = m + (a-m)/n
//
//
//Bei jeder neuen Berechnung wird der FC-ENO Ausgang HIGH
//
//
//AUTOR: Stefan Maag, Dipl.-Ing. (FH) Elektrotechnik
//DATUM: 9/2005
//INTERNET: www.maagic7.de
//
//AENDERUNGSVERMERKE:
//--------------------------------------------------------------------------------
//DATUM        NAME            AENDERUNG
//--------------------------------------------------------------------------------
//
//--------------------------------------------------------------------------------
//
//HINWEISE:
AUTHOR : 'S.Maag'
FAMILY : Maagic7
VERSION : 0.1


VAR_INPUT
  CALC : BOOL ;	//Neuen Mittelwert bilden
  RESET : BOOL ;	//RESET
  VALUE : DINT ;	//Eingangswert
END_VAR
VAR_OUTPUT
  M_DINT : DINT ;	//Mittelwert im DINT-Format
END_VAR
VAR_IN_OUT
  M_REAL : REAL ;	//Mittelwert im REAL-Format
  N : DINT ;	//Anzahl der bereits verrechneten Werte
END_VAR
VAR_TEMP
  diff : REAL ;
END_VAR
BEGIN
NETWORK
TITLE =



NETWORK
TITLE =RESET

      UN    #RESET;
      SPB   NE2;

      L     0; // Rücksetzen
      T     #N; // Anzahl verrechneter Werte
      T     #M_DINT; // Mittelwert DINT

      L     0.000000e+000; // Mittelwert löschen
      T     #M_REAL;

NE2:  NOP   0;

NETWORK
TITLE =

      U     #CALC;
      SAVE  ;
      SPB   CLC;
      SPA   OUT;


NETWORK
TITLE =Anzahl der Verrechneten Werte erhöhen

CLC:  L     #N;
      +     L#1;
      T     #N;

NETWORK
TITLE =neuen Mittelwert berechnen
//
//neuesMittel = Mittelwert + (Eingangswert - Mittelwert) / AnzahlWerte
      L     #VALUE; // Eingangswert
      DTR   ; // in Real wandeln
      L     #M_REAL; // und vom aktuellen Mittelwert abziehen
      -R    ; // =(Eingangswert - Mittelwert)
      T     #diff;
      L     #N;
      DTR   ;
      /R    ; // = (Eingangswert - Mittelwert)/AnzahlWerte
      L     #M_REAL;
      +R    ;
      T     #M_REAL; // neuer Mittelwert



NETWORK
TITLE =Mittelwert als DINT ausgeben

OUT:  L     #M_REAL;
      RND   ; // in Ganzzahl wandeln
      T     #M_DINT;

END_FUNCTION

FUNCTION "m7b_RAMPE_LIN_min" : VOID
TITLE =Linear-Rampen-Generator mit MaxBegrenzung für Hand und Auto
//Generiert eine lineare Rampe zwischen den Geschwindigkeiten MIN und MAX.
//Bei einer Entfernung = RampenDistanz wird die Rampe eingeleitet.
//Bei einer Entfernung = Vk_MinSpeed erreicht die Rampe Speed_min
//
//AUTOR: Stefan Maag, Dipl.-Ing. (FH) Elektrotechnik
//DATUM: 3/2003
//INTERNET: www.maagic7.de
//
//AENDERUNGSVERMERKE:
//--------------------------------------------------------------------------------
//DATUM        NAME          AENDERUNG
//--------------------------------------------------------------------------------
//12.09.2007   S. Maag       Vorkontakt bei Berechnung der Rampenlänge
//                           berücksichtigt. Nun glatter Übergang bei erreichen
//                           des Vorkontaktes. (NW3: RAMP:)
//
//20.04.2009   S. Maag       FC-ENO:= True, wenn innerhalb der Rampe
//--------------------------------------------------------------------------------
//
//HINWEISE:
AUTHOR : 'S.Maag'
FAMILY : Maagic7
VERSION : 0.1


VAR_INPUT
  VK_MinSpeed : DINT ;	//Vorkontakt für Fahrt mit Minimalgeschwindigkeit
  Speed_min : INT ;	//Geschwindigkeit minimal
  Speed_max : INT ;	//Geschwindigkeit maximal
  RampenDistanz : DINT ;	//Positionsdistanz, ab der mit der Rampe begonnen wird
  SW_Pos : DINT ;	//Sollwert Position
  IW_Pos : DINT ;	//Istwert Position
END_VAR
VAR_OUTPUT
  Speed : INT ;	//Solwert Geschwindigkeit
END_VAR
VAR_TEMP
  SPEED_DIFF : INT ;
  POS_DIFF : DINT ;
  RAMP_LENGTH : DINT ;
END_VAR
BEGIN
NETWORK
TITLE =Geschwindigkeitsbereich, Geschwindigkeitsdifferenz


      L     #Speed_max; // Maximalgeschwindigkeit
      L     #Speed_min; // Minimalgeschwindigkeit
      -I    ;
      T     #SPEED_DIFF; // Geschwindigkeitsbereich absolut

NETWORK
TITLE =Positionsdifferenz positiv: ABS(Soll - Ist)

      L     #SW_Pos; // Soll-Position
      L     #IW_Pos; // Ist-Position
      -D    ; // Positionierabstand
      SPP   PLUS; // positiven Wert erzeugen
      NEGD  ;
PLUS: T     #POS_DIFF; // Positionierdifferenz
      L     #VK_MinSpeed; // Vorkontakt für Fahrt mit Minimalgeschw.
      <D    ;
      SPB   MIN; // Minimalgeschw. laden

      TAK   ; // POS_DIFF in Akku 1 zurück
      L     #RampenDistanz; // Rampendistanz
      <=D   ; // Wenn Pos_Diff<RampenDist
      SAVE  ;
      SPB   RAMP; // -> innerhalb der Rampe; Rampe generieren

      L     #Speed_max; // Maximalgeschwindigkeit
      SPA   SAVE;

MIN:  SET   ;
      SAVE  ;
      CLR   ;

      L     #Speed_min; // andernfalls die Minimalgeschwindigkeit
      SPA   SAVE; // als SpeedAkt speichern
NETWORK
TITLE =Rampe generieren:
//SpeedDiff = SpeedMax - SpeedMin  :  Geschwindigkeitsbereich
//
//V(RAMPE) = SpeedDiff * (PosDiff / RampenDistanz) + SpeedMin
// Rampe generieren wird nur aufgerufen, wenn man sich innerhalb der
// Rampendistanz befindet, sonst wird SpeedMin ausgegeben
// 12.09.2007: Vorkontakt bei Berechnung der Rampenlänge berücksichtigt

RAMP: L     #RampenDistanz; // Rampendistanz (Eingang)
      L     #VK_MinSpeed; // Vorkontakt Minimalgeschwindigkeit
      -D    ;
      T     #RAMP_LENGTH; // berechnete Rampenlänge bis Vorkontakt

      L     #POS_DIFF; // Positionierdifferenz
      DTR   ; // nach REAL
      L     #RAMP_LENGTH; // berechnete RampenDistanz
      DTR   ; // nach REAL
      /R    ; // PosDiff / RampenDistanz
      L     #SPEED_DIFF; // SpeedDiff
      ITD   ; // nach DINT
      DTR   ; // nach REAL
      *R    ;
      RND   ; // nach DINT
      L     #Speed_min; // SpeedMin
      ITD   ; // nach DINT
      +D    ;
      L     DW#16#FFFF; // nach INT
      UD    ; // Aktueller Speed als INT in AKKU1

NETWORK
TITLE =nun noch auf Maximalwert bei Hand oder Auto begrenzen

SAVE: L     #Speed_max; // Speed max
      >I    ; // Wenn SpeedAkt >  MaxSpeed,
      SPB   SAV0; // dann MaxSpeed speichern
      TAK   ; // sonst SpeedAkt zurück in Akku1
SAV0: T     #Speed; // Speed speichern

END_FUNCTION

FUNCTION "m7b_POSITONIEREN" : VOID
TITLE =Positionierrichtung Achse ermitteln. Position ok ausgeben
//Dieser FC ermittelt die Positonierrichtung von Achsen (vorw./rückw.)
//
//TOL_POS : Ist die zuslässige Positionsdifferenz, ab der die Achse zum
//          nachpositionieren anfängt
//
//TOL_POS_OK : Ist die zulässige Toleranz bis zu der gemeldet wird, dass
//             die Achse im gültigen Positiosfenster steht
//
//AUTOR: Stefan Maag, Dipl.-Ing. (FH) Elektrotechnik
//DATUM: 8/2003
//INTERNET: www.maagic7.de
//
//AENDERUNGSVERMERKE:
//--------------------------------------------------------------------------------
//DATUM        NAME        AENDERUNG
//--------------------------------------------------------------------------------
//21.04.2009   S.Maag      TOL_POS auf ENO-Ausgang, damit kann verzögert dann
//                         die Freigabe für den Positionier-FB gelöscht werden
//--------------------------------------------------------------------------------
//
//HINWEISE:
AUTHOR : 'S.Maag'
FAMILY : Maagic7
VERSION : 0.1


VAR_INPUT
  FRG : BOOL ;	//Freigabe
  SOLL : DINT ;	//Sollwert
  IST : DINT ;	//Istwert Achse
  TOL_POS_OK : DINT ;	//Toleranz für Position ok Meldung
  TOL_POS : DINT ;	//Toleranz Posiitionierung Achse
END_VAR
VAR_OUTPUT
  PLUS : BOOL ;
  MINUS : BOOL ;
  POS_OK : BOOL ;
END_VAR
BEGIN
NETWORK
TITLE =Postion Achse prüfen, Positionsdifferenz

      L     #SOLL; // aktuelle Sollposition
      L     #IST; // aktuelle Istposition
      -D    ; // Positionierdifferenz
      SPP   PLUS;
      NEGD  ; // nach positiv

PLUS: L     #TOL_POS_OK; // Toleranz für Position ok
      <D    ;
      =     #POS_OK; // Ausgang Position ok

      TAK   ; // Positionsdifferenz in AKKU1
      L     #TOL_POS; // Toleranz für Positionierung
      <D    ;
      SAVE  ;
      SPB   STOP; // Innerhalb Toleranz, dann Stop

NETWORK
TITLE =FREIGABE

      UN    #FRG; // keine Freigabe, dann Stop
      SPB   STOP;

NETWORK
TITLE =Postionierrichtung vorw. oder rückw.

      L     #SOLL; // Soll
      L     #IST; // IST
      >D    ;
      SPB   VW; // Soll > Ist, dann vw
      SPA   RW; // sonst rw
NETWORK
TITLE =Richtungsausgänge setzen

STOP: R     #PLUS;
      R     #MINUS;
      BEA   ;

VW:   R     #MINUS;
      S     #PLUS;
      BEA   ;

RW:   R     #PLUS;
      S     #MINUS;
      BE    ;
END_FUNCTION

FUNCTION "m7b_SPEED_SELECT" : VOID
TITLE =Speed auswählen
//AUTOR: Stefan Maag, Dipl.-Ing. (FH) Elektrotechnik
//DATUM: 8/2003
//INTERNET: www.maagic7.de
//
//AENDERUNGSVERMERKE:
//--------------------------------------------------------------------------------
//DATUM        NAME        AENDERUNG
//--------------------------------------------------------------------------------
//13.03.2020   S.Maag      Baustein aus Library entfernt, wird druch
//                         FC113/114 MUX_INT ersetzt
//24.04.2009   S.Maag      EN0 := Signal Wert selektiert
//                               (S1 | S2 | S3)  AND ENABLE
//--------------------------------------------------------------------------------
//
//HINWEISE:
AUTHOR : 'S.Maag'
FAMILY : Maagic7
VERSION : 0.1


VAR_INPUT
  S1 : BOOL ;	//Auswahl Speed 1 (1-te Priorität)
  S2 : BOOL ;	//Auswahl Speed 2 (2-te Priorität)
  S3 : BOOL ;	//Auswahl Speed 3 (3-te Priorität)
  FRG : BOOL ;
  SPEED_1 : INT ;
  SPEED_2 : INT ;
  SPEED_3 : INT ;
END_VAR
VAR_OUTPUT
  SPEED : INT ;
END_VAR
BEGIN
NETWORK
TITLE =

      UN    #FRG; // keine Freigabe, dann 0 ausgeben
      SPB   STOP;

      U     #S1;
      SPB   S1;

      U     #S2;
      SPB   S2;

      U     #S3;
      SPB   S3;
      SPA   STOP;

S1:   L     #SPEED_1;
      SPA   SAVE;

S2:   L     #SPEED_2;
      SPA   SAVE;

S3:   L     #SPEED_3;
      SPA   SAVE;

STOP: CLR   ; // EN0-Ausgang =0, da Stopp
      SAVE  ;
      L     0;
      T     #SPEED;
      BEA   ;

SAVE: T     #SPEED;
      SAVE  ;
END_FUNCTION

FUNCTION "m7b_READ_SSI_ENCODER" : VOID
TITLE =SSI-Encoder einlesen: Position mit Auflösung & 0-Pkt-Korrektur
//[IN]
//PED_IN         Perepherie-Kanal SSI-ENCODER z.B. PED256
//Encoder_Bits   Anzahl der Bits, die Encoder verarbeitet, meist 24 oder 25.
//               Diese Angabe ist vor allem für invertierte Drehrichtung
//               wichtig, da sonst die hohen nicht belegten Bits des Encoders
//               immer 1 sind, was einen grossen negtiven Wert bedeuted.
//
//FKT_AUFL       Faktor für Endoderauflösung
//O_Pkt_Korr     0-Punkt Korrekturwert, Wert wird addiert
//INV            Drehrichtung invertieren
//
//[OUT]
//POS_DINT       Position als DINT-Wert 32 Bit
//POS_INT        Position als INT-Wert 16 Bit
//
//AUTOR: Stefan Maag, Dipl.-Ing. (FH) Elektrotechnik
//DATUM: 7/2008
//INTERNET: www.maagic7.de
//
//AENDERUNGSVERMERKE:
//--------------------------------------------------------------------------------
//DATUM      NAME     AENDERUNG
//--------------------------------------------------------------------------------
//
//--------------------------------------------------------------------------------
//
//HINWEISE:
AUTHOR : 'S.Maag'
FAMILY : Maagic7
VERSION : 0.1


VAR_INPUT
  PED_IN : DWORD ;	//Perepherie-Kanal SSI-ENCODER z.B. PED256
  EncoderBits : INT ;	//Anzahl der Bits, die Encoder verarbeitet, meist 24 oder 25
  FKT_AUFL : REAL ;	//Faktor Auflösung, wird multipliziert
  O_Pkt_Korr : DINT ;	//0-Punkt Korrekturwert, Wert wird addiert
  INV : BOOL ;	//Drehrichtung invertieren
END_VAR
VAR_OUTPUT
  POS_DINT : DINT ;	//Position als DINT-Wert 32 Bit
  POS_INT : INT ;	//Position als INT-Wert 16 Bit
END_VAR
VAR_TEMP
  MASKE : DWORD ;	//Bitmaske zur verarbeitender Bits des Encoder, meist nur 24Bit
  Bits : INT ;
END_VAR
BEGIN
NETWORK
TITLE =Bitmaske der vom Geber verarbeiteten Anzahl der Bits erzeugen

      L     #EncoderBits; // Anzahl der vom Encoder verarbeitetn Bits max. 32
      DEC   1; // umrechnen auf 0..31 durch abziehen von 1
      L     2#11111; // Auf 5 Bit := 0..31
      UW    ; // begrenzen
      L     31; // max. zu verarbeitender Bitwert in Akku 1
      TAK   ; // vom Encoder max. verarbeiter Bitwert 0..31 in Akku 1 zurück
      -I    ; // Vom Encoder wengier als verarbeitet Bits
      L     DW#16#FFFFFFFF; // 32 Bits auf 1 := Maske bei 32 verarbeitetn Bits
      SRD   ; // Maske um Differenz der Bits in Akku2-LL verschieben
      T     #MASKE; // = Maske der vom Encoder verarbeiteten Bits
NETWORK
TITLE =Encoderwert mit Auflösung und 0-Punkt-Korrektur berechnen

      L     #PED_IN; // Wert von Encoder
      UN    #INV; // Drehrichtung invertieren ?
      SPB   calc; // wenn nein, dann berechnen
      NEGD  ; // Wert invertieren
calc: L     #MASKE; // Geber hat meist keine 32Bit, Rest ausblenden
      UD    ; // sonst sind bei invertierter Messrichtung die höchsten Bits immer 1
      DTR   ; // wandeln nach Real
      L     #FKT_AUFL; // Faktor für Geberanpassung
      *R    ;
      RND   ; // in DINT zurückwandeln
      L     #O_Pkt_Korr; // Korrekturwert für 0-Punktverschiebung
      +D    ;
      T     #POS_DINT; // Istwert Encoder 32 Bit
      T     #POS_INT; // Istwert Encoder 16 Bit
NETWORK
TITLE =FC-ENO = HIGH

      SET   ;
      SAVE  ;
      CLR   ;

END_FUNCTION

FUNCTION "m7b_ENCODER_KORR" : VOID
TITLE =Encoderwerte: Position mit Auflösung & 0-Pkt-Korrektur
//[IN]
//ENCODER        Roh-Wert des Encoders
//Encoder_Bits   Anzahl der Bits (1..32), die verarbeitet werden sollen.
//               Bei SSI-Encodern sind dies meist 24;25 Bits.
//               Diese Angabe ist vor allem für invertierte Drehrichtung
//               wichtig, da sonst die hohen nicht belegten Bits des Encoders
//               immer 1 sind, was einen grossen negtiven Wert bedeuted.
//FKT_AUFL       Faktor für Endoderauflösung
//O_Pkt_Korr     0-Punkt Korrekturwert, Wert wird addiert
//INV            Drehrichtung invertieren
//
//[OUT]
//POS_DINT       Position als DINT-Wert 32 Bit
//POS_INT        Position als INT-Wert 16 Bit
//
//AUTOR: Stefan Maag, Dipl.-Ing. (FH) Elektrotechnik
//DATUM: 7/2008
//INTERNET: www.maagic7.de
//
//AENDERUNGSVERMERKE:
//--------------------------------------------------------------------------------
//DATUM      NAME     AENDERUNG
//--------------------------------------------------------------------------------
//
//--------------------------------------------------------------------------------
//
//HINWEISE:
AUTHOR : 'S.Maag'
FAMILY : Maagic7
VERSION : 0.1


VAR_INPUT
  ENCODER : INT ;	//Perepherie-Kanal SSI-ENCODER z.B. PED256
  EncoderBits : INT ;	//Anzahl der Bits, die Encoder verarbeitet (1..32), meist 24 oder 25
  FKT_AUFL : REAL ;	//Faktor Auflösung, wird multipliziert
  O_Pkt_Korr : DINT ;	//0-Punkt Korrekturwert, Wert wird addiert
  INV : BOOL ;	//Drehrichtung invertieren
END_VAR
VAR_OUTPUT
  POS_DINT : DINT ;	//Position als DINT-Wert 32 Bit
  POS_INT : INT ;	//Position als INT-Wert 16 Bit
END_VAR
VAR_TEMP
  MASKE : DWORD ;	//Bitmaske zur verarbeitender Bits des Encoder, meist nur 24Bit
  Bits : INT ;
END_VAR
BEGIN
NETWORK
TITLE =Bitmaske der vom Encoder verarbeiteten Anzahl der Bits erzeugen

      L     #EncoderBits; // Anzahl der vom Encoder verarbeitetn Bits max. 32
      DEC   1; // umrechnen auf 0..31 durch abziehen von 1
      L     2#11111; // Auf 5 Bit := 0..31
      UW    ; // begrenzen
      L     31; // max. zu verarbeitender Bitwert in Akku 1
      TAK   ; // vom Encoder max. verarbeiter Bitwert 0..31 in Akku 1 zurück
      -I    ; // Vom Encoder weniger als verarbeitete Bits
      L     DW#16#FFFFFFFF; // 32 Bits auf 1 := Maske bei 32 verarbeitetn Bits
      SRD   ; // Maske um Differenz der Bits in Akku2-LL verschieben
      T     #MASKE; // = Maske der vom Encoder verarbeiteten Bits
NETWORK
TITLE =Encoderwert mit Auflösung und 0-Punkt-Korrektur berechnen

      L     #ENCODER; // Wert von Encoder
      UN    #INV; // Drehrichtung invertieren ?
      SPB   calc; // wenn nein, dann berechnen
      NEGD  ; // Wert invertieren
calc: L     #MASKE; // Geber hat meist keine 32Bit, Rest ausblenden
      UD    ; // sonst sind bei invertierter Messrichtung die höchsten Bits immer 1
      DTR   ; // wandeln nach Real
      L     #FKT_AUFL; // Faktor für Geberanpassung
      *R    ;
      RND   ; // in DINT zurückwandeln
      L     #O_Pkt_Korr; // Korrekturwert für 0-Punktverschiebung
      +D    ;
      T     #POS_DINT; // Istwert Encoder 32 Bit
      T     #POS_INT; // Istwert Encoder 16 Bit
NETWORK
TITLE =FC-ENO = HIGH

      SET   ;
      SAVE  ;
      CLR   ;

END_FUNCTION

FUNCTION "m7b_TACHO" : VOID
TITLE =Tacho: (zurückgelegter Weg je Zeiteinheit)
//AUTOR: Stefan Maag, Dipl.-Ing. (FH) Elektrotechnik
//DATUM: 5/2003
//INTERNET: www.maagic7.de
//
//Dieser FC ermittelt den zurückgelegten Weg je Zeiteinheit.
//Der Weg wird absolut (immer positiv) ermittelt und entspricht somit der
//Geschwindigkeit.
//Zusätzlich werden die Richtungen POSITIV und NEGAIV als extra Signal ausgegeben.
//Ist keines der beiden Signale aktiv, so steht die Achse
//
//AENDERUNGSVERMERKE:
//--------------------------------------------------------------------------------
//DATUM        NAME            AENDERUNG
//--------------------------------------------------------------------------------
//30.10.2017   S.Maag         io_SpeedPulse von INT auf DINT geaendert
//                            INT macht hier keinen Sinn!
//
//17.11.2006   S.Maag         FC getestet
//                            FC-ENO-Ausgang = Antrieb läuft; hinzugefügt
//--------------------------------------------------------------------------------
//
//HINWEISE:
AUTHOR : 'S.Maag'
FAMILY : Maagic7
VERSION : 0.1


VAR_INPUT
  ENCODER : DINT ;	//Positionswert des Encoders
  TA_IMP : BOOL ;	//Abtastimpuls, Impuls (1Zyklus)
  FRG : BOOL ;	//Freigabe, Start
END_VAR
VAR_OUTPUT
  POSITIV : BOOL ;	//Drehrichtung positiv
  NEGATIV : BOOL ;	//Drehrichtung negativ
END_VAR
VAR_IN_OUT
  io_dSpeedPulse : DINT ;	//Geschwindigkeit als Positionswerte je TriggerEreignis
  memENCODER : DINT ;	//Speicherung der Encoder StartPosition
  memByte : BYTE ;	//Hilfspeicher BYTE
END_VAR
VAR_TEMP
  tmpStart : BOOL ;
  tmpPositiv : BOOL ;
  tmpNegativ : BOOL ;
  LB_3 : BOOL ;
  LB_4 : BOOL ;
  LB_5 : BOOL ;
  LB_6 : BOOL ;
  LB_7 : BOOL ;
END_VAR
BEGIN
NETWORK
TITLE =

      L     #memByte; // Hilfword für Signalspeicherung
      T     LB     0; // in Lokaldatenbereich, wegen Bitadressierung
NETWORK
TITLE =START-Eingang prüfen

      UN    #FRG; // Wenn nicht gestartet, dann
      R     #tmpStart; // HM Start löschen
      BEB   ;
NETWORK
TITLE =Start-Ereignis verarbeiten

      U     #tmpStart;
      SPB   NWE;

      S     #tmpStart; // HM gestartet
      L     #ENCODER; // akt. EncoderWert
      T     #memENCODER; // als Vergleich speichern
      SPA   END;
NWE:  NOP   0;

NETWORK
TITLE =Trigger-Ereignis : Speed ermitteln

      UN    #TA_IMP; // Wenn Trigger-Ereignis eintritt,
      SPB   END;

      L     #memENCODER; // StartPos Encoder
      L     #ENCODER; // akt. EncoderPos
      T     #memENCODER; // als neue StartPos speichern
      -D    ; // zurückgelegten Weg ermitteln
      U     >0; // Wegdifferenz <0 (da memENC-ENC)
      =     #tmpNegativ; // = Drehrichtung negativ
      U     <0; // Wegdifferenz >0 (da memENC-ENC)
      =     #tmpPositiv; // = Drehrichtung positiv
      SPP   PLUS;
      NEGD  ;
PLUS: T     #io_dSpeedPulse; // SPEED = WEG / ZeitEinheit

NETWORK
TITLE =Richtungsausgänge Ausgeben
//die Richtungsausgänge müssen über den Umweg eines statischen Hilfsspeichers
//immer Ausgegeben werden. Bei direkter Ausgabe hätten sie einen nicht
//definierten
//Zustand, da die Ausgabe im obigen NW nur mit Auftreten eines Impulses erfolgt
END:  U     #tmpNegativ;
      =     #NEGATIV;
      U     #tmpPositiv;
      =     #POSITIV;

NETWORK
TITLE =FC-ENO Ausgang = Antrieb läuft, RUN

      O     #tmpNegativ;
      O     #tmpPositiv;
      SAVE  ;
      CLR   ;

NETWORK
TITLE =Bitadressierte Signale aus Lokaldatenbereich wieder speichern

      L     LB     0; // Lokaldatenword
      T     #memByte; // nach Singnalspeicher

END_FUNCTION

FUNCTION "m7b_WEG_ZAEHLER" : VOID
TITLE =Weg-Zähler (km Zähler)
//Dieser FC arbeitet als Weg-Zähler, vergleichbar einem km-Zähler.
//
//IN: ENDODER: Positionswert des zu zählenden Encoders
//IN: INKR   : Anzahl der Weginkremente, die jeweils eine Zähleinheit bilden
//IN: FRG    : Zählfreigabe; Zählvorgang an der akt. EncoderPos. beginnen
//IN: RICHTUNG: hiermit kann die Zählrichtung für den Weg angebeben werden 0:+/1:-
//
//Der Baustein verfügt über eine integrierte Fehlerkorrektur: D.h. es soll z.B.
//in einer Teilung von je 100 INKR gezählt werden. Dabei kommt es vor, bedingt
//durch SPS Zykluszeit usw., das das Zählerereignis erst bei einem Weg von z.B.
//105 INKR bearbeitet wird. Dies wird korrigiert, indem beim nächsten Mal die
//Soll-Inkremente dann auf 95 festgelegt werden usw. Dies verhindert einen sich
//aufschaukelden Fehler!
//
//AUTOR: Stefan Maag, Dipl.-Ing. (FH) Elektrotechnik
//DATUM: 3/2003
//INTERNET: www.maagic7.de
//
//AENDERUNGSVERMERKE:
//--------------------------------------------------------------------------------
//DATUM        NAME            AENDERUNG
//--------------------------------------------------------------------------------
//
//--------------------------------------------------------------------------------
//
//HINWEISE:
AUTHOR : 'S.Maag'
FAMILY : Maagic7
VERSION : 0.1


